	VH11.IdXML					:=	'1';
	VH11.TagXML					:=	4;
	VH11.DEF_On.IdXML			:=	'3';
	VH11.DEF_On.TagXML			:=	2;
	VH11.DEF_Off.IdXML			:=	'3';
	VH11.DEF_Off.TagXML			:=	4;
	VH11.DEF_Sensor.IdXML		:=	'3';
	VH11.DEF_Sensor.TagXML		:=	13;
	VH11.DEF_On_Imposs.IdXML	:=	'3';
	VH11.DEF_On_Imposs.TagXML	:=	6;
	VH11.DEF_Off_Imposs.IdXML	:=	'3';
	VH11.DEF_Off_Imposs.TagXML	:=	9;
	VH11.DEF_Off_auto.IdXML		:=	'3';
	VH11.DEF_Off_auto.TagXML	:=	11;

	VS11.IdXML					:=	'1';
	VS11.TagXML					:=	3;

	VINT.IdXML					:=	'1';
	VINT.TagXML					:=	1;
	VINT.DEF_On.IdXML			:=	'3';
	VINT.DEF_On.TagXML			:=	2;
	VINT.DEF_Off.IdXML			:=	'3';
	VINT.DEF_Off.TagXML			:=	4;
	VINT.DEF_Sensor.IdXML		:=	'3';
	VINT.DEF_Sensor.TagXML		:=	13;
	VINT.DEF_On_Imposs.IdXML	:=	'3';
	VINT.DEF_On_Imposs.TagXML	:=	6;
	VINT.DEF_Off_Imposs.IdXML	:=	'3';
	VINT.DEF_Off_Imposs.TagXML	:=	9;
	VINT.DEF_Off_auto.IdXML		:=	'3';
	VINT.DEF_Off_auto.TagXML	:=	11;


(* Gestion FM et FD régénération*)
FM_REGEN(CLK:=PS11.STATE_Regen);
FD_REGEN(CLK:=PS11.STATE_Regen);
END_ACTION

END_FUNCTION_BLOCK

// ---- POUs/Fonction/FONCTIONS PUISSANCE/BLOCK_CPT_USURE_OLD.TcPOU
FUNCTION_BLOCK BLOCK_CPT_USURE_OLD

VAR_INPUT
	I_Machine_prod:			BOOL;		(*Indicateur de machine en process*)
	I_EVAP_ON:	BOOL;			(*Indicateur d'évaporation en cours*)
END_VAR

VAR
	O_Rapport:					BOOL;		(*demande d'édition du rapport de consommation, c'est l'outil externe qui la fait retomber*)

	FM_Prod:					R_TRIG;		(*Front montant de debut de prod*)
	FM_Layer_Load_Ok:			R_TRIG;		(*Front montant de chargement couche ok*)
	FM_Layer:					R_TRIG;		(*Front montant début évaporation*)
	FD_Prod:					F_TRIG;		(*Front descendant de fin de prod*)

	FD_O_Rapport:				F_TRIG;		(*Front descendant de demande d'édition du rapport*)
	FD_Layer:					F_TRIG;		(*Front descendant de fin de couche*)

	VAR_New_File:				BOOL;		(*Indique si un nouveau fichier doit être créee*)


END_VAR

VAR_OUTPUT
	(*Données du rapport*)
	STATE_User_Login:			STRING[30];	(*Login user ayant lancé la prod*)
	STATE_User_Name:			STRING[30];	(*Nom user ayant lancé la prod*)
	STATE_User_First:			STRING[30];	(*Prénom user ayant lancé la prod*)

	STATE_Process_Name:		STRING;		(*Nom du procédé lancé*)
	STATE_Date_Deb:			DT;			(*Debut du process*)
	STATE_Date_Fin:				DT;			(*Fin du process*)


	STATE_Config:			STRING;		(*Configuration utilisé*)
	STATE_Crucible:			USINT;		(*Numéro du creuset utilisé*)
	STATE_Material:				STRING;		(*Nom du matériau utilisé*)

	STATE_THICK_Consigne:			REAL;	(*Epaisseur saisie par l'utilisateur au début de la recette*)
	STATE_THICK_Obtenue:			REAL;	(*Epaisseur obtenue en fin de couche ou sur arrêt procédé*)

	STATE_Date_Deb_Evap:		DT;		(*Début d'évaporation*)
	STATE_Date_Fin_Evap:		DT;		(*Fin évaporation*)
	STATE_Temps_Depot:			INT;	(*Temps du dépôt*)

END_VAR

(*Gestion des fronts*)
FM_Prod(clk := I_Machine_prod);
FD_Prod(clk := I_Machine_prod);

FM_Layer(clk := I_EVAP_ON );
FD_Layer(clk := I_EVAP_ON);

FD_O_Rapport(clk := O_Rapport);

(*Remise à 0 des valeurs*)
IF FD_O_Rapport.Q THEN
	STATE_Config				:= '';
	STATE_Crucible				:= 0;
	STATE_Material				:= '';
	STATE_THICK_Consigne		:= 0;
	STATE_THICK_Obtenue			:= 0;
END_IF

(*Enregistrement des données en début de process*)
IF FM_Prod.Q THEN
	VAR_New_File					:=	TRUE;
	STATE_User_Login				:=	PRG_USER.ACTU_USER.LOGIN;
	STATE_User_Name				:=	PRG_USER.ACTU_USER.NOM;
	STATE_User_First				:=	PRG_USER.ACTU_USER.PRENOM;

	STATE_Process_Name			:=	EXECPROC.PRM_PROCESS;
	STATE_Date_Deb				:=	PRG_SEC._date;

END_IF


(*Enregistrement des données liées à l'empilement*)
IF FM_Layer_Load_Ok.Q THEN
	STATE_Config				:= PRG_MOUVEMENT_PS.STATE_Dome_Type;
	STATE_Crucible				:= PRG_EVAP.EVAPS1.PRM_NCR;
	STATE_Material				:= PRG_EVAP.CRUCIBLE1.PRM_MAT[STATE_Crucible];
	STATE_THICK_Consigne		:= MAIN.STEP_EMPILEMENT.PRM_EPAISSEUR;
END_IF


(*Enregistrements des données en début de couche*)
IF FM_Layer.Q THEN
	STATE_Date_Deb_Evap				:= PRG_SEC._date;
END_IF


(*Enregistrements des données en fin de couche*)
IF FD_Layer.Q THEN
	STATE_Date_Fin_Evap				:= PRG_SEC._date;
	STATE_THICK_Obtenue			:= MAIN.STEP_EMPILEMENT.STATE_RATE_AGREGATE;

		(*Levée du bit de demande de création d'un nouveau fichier*)
		O_Rapport					:=	TRUE;

END_IF


IF FD_Prod.Q THEN
	STATE_Date_Fin	:= PRG_SEC._date;

		(*Levée du bit de demande de création d'un nouveau fichier*)
		O_Rapport					:=	TRUE;

END_IF

END_FUNCTION_BLOCK

// ---- POUs/Fonction/FONCTIONS SERVITUDES/BLOCK_LIGNE_REF_FLOWTEMP.TcPOU
FUNCTION_BLOCK BLOCK_LIGNE_REF_FLOWTEMP

(* Fonction de gestion d'une ligne d'eau avec débitmètre SV4200 (Vanne avec ou sans débitmètre*)

(****************historique des versions*****************************)
(* Version 1-0 - GV - 07/2023 - VERSION INITIALE - 13905*)
(********************************************************************)

VAR_INPUT
	RESET:					BOOL;
	MANUAL:					BOOL;			(* ~ (OPC : 1 : available for OPC-clients) *)
	DEx:					BLOCK_SV4200;

	CO_On:					BOOL;								(*commande de marche*)
                                                                
	I_Cond_need_Ref:		BOOL;								(*condition qui necessite le refroidissement*)
	I_inhibe_surv_ref:		BOOL;								(*Condition d'inhibition de la surveillance du débit*)
	I_Cond_ref_Ok:			BOOL;								(*Condition de validation du bon refroidissment (Temp, ...) *)
                                                                
	VEx:					BLOCK_ACTUATOR;						(*vanne d'eau simple*)
                                                                
	DEF_Ref:				PRCDEF;								(*défaut de refroidissement*)
	DEF_Dex:				PRCDEF;								(*défaut de fonctionnement du débitmètre*)
	                                                            
	DEF_Low_Flow:			PRCDEF;								(*défaut débit insuffisant*)
	DEF_High_Flow:			PRCDEF;								(*défaut débit trop important*)
	DEF_Low_Temp:			PRCDEF;								(*défaut température trop basse*)
	AL_High_Temp:			PRCDEF;								(*alarme température trop haute*)
	DEF_High_Temp:			PRCDEF;								(*défaut température trop haute*)
END_VAR

VAR_INPUT PERSISTENT
	CONF_NO_DexT:			BOOL;								(*option pas de débitmètre*)
	CONF_TIM_OFF:			TIME;								(* ~ (OPC : 1 : available for OPC-clients) *)		(*temps entre la perte de la condition absolue de refroidissement
																					et la fermeture de la vanne d'eau*)
	CONF_No_Def_Dex:		BOOL;													(*pas de surveillance du défaut de fermeture de la vanne*)

	CONF_Eau_chaude:		BOOL;			(*ligne d'eau raccordée à un circuit eau chaude/froide*)
	
	CONF_Min_Flow:			REAL;			(*débit minimum*)
	CONF_Max_Flow:			REAL;			(*Débit maximum*)
	CONF_Min_Temp:			REAL;			(*Température minimum*)
	CONF_Max_Temp:			REAL;			(*Température maximum pour défaut*)	
	CONF_Max_Temp_AL:		REAL;			(*Température maximum pour alarme*)

	(*Entité*)
	IsAssembly:				BOOL;			(*entité : assemblage*)
	IdXML:					STRING;			(*nom entité : identifiant pour recherche dans dico*)
	TagXML:					UINT;			(*nom entité : identifiant pour recherche dans dico*)
	IdParent:				STRING;			(*MNEMO de l'appelant*)
	MNEMO:					STRING;			(*MNEMO de l'entité*)
	MNEMO_Dex:				STRING;			(*MNEMO du débitmètre*)
END_VAR

VAR_OUTPUT
	STATE_Ok:				BOOL;			(* ~ (OPC : 1 : available for OPC-clients) *)		(*refroidissement ok*)
	STATE_Ar:				BOOL;			(* ~ (OPC : 1 : available for OPC-clients) *)		(*refroidissement à l'arrêt*)
	STATE_NOk:				BOOL;			(* ~ (OPC : 1 : available for OPC-clients) *)		(*refroidissement à l'arrêt*)
	STATE_DexT:				BOOL;			(* ~ (OPC : 1 : available for OPC-clients) *)		(*seuil débitmètre*)
END_VAR

VAR
	TIMER_OFF:					TON;
	VAR_Etape:					USINT;															(*Etape du grafcet de gestion de la servitudes*)
	VAR_DExT:					BOOL;
END_VAR

Def_Ref.IdXML				:=	'8';
Def_Ref.TagXML				:=	1;

DEF_Dex.IdXML				:=	'8';
DEF_Dex.TagXML				:=	2;

DEF_Low_Flow.IdXML			:=	'8';
DEF_Low_Flow.TagXML			:=	15;
DEF_High_Flow.IdXML			:=	'8';
DEF_High_Flow.TagXML		:=	16;
DEF_Low_Temp.IdXML			:=	'8';
DEF_Low_Temp.TagXML			:=	17;
DEF_High_Temp.IdXML			:=	'8';
DEF_High_Temp.TagXML		:=	18;
AL_High_Temp.IdXML			:=	'8';
AL_High_Temp.TagXML			:=	18;
AL_High_Temp.Groupe			:=	1;

VEx.IdParent				:=	MNEMO;
VEx.IdXML					:=	'1';
VEx.TagXML					:=	1;
VEx.DEF_Off_auto.IdXML		:=	'3';
VEx.DEF_Off_auto.TagXML		:=	11;
VEx.DEF_Off_Imposs.IdXML	:=	'3';
VEx.DEF_Off_Imposs.TagXML	:=	9;
VEx.DEF_On_Imposs.IdXML		:=	'3';
VEx.DEF_On_Imposs.TagXML	:=	6;
VEx.DEF_On.IdXML			:=	'3';
VEx.DEF_On.TagXML			:=	2;
VEx.DEF_Off.IdXML			:=	'3';
VEx.DEF_Off.TagXML			:=	4;
VEx.DEF_Sensor.IdXML		:=	'3';
VEx.DEF_Sensor.TagXML		:=	13;
	
(*Débitmètre*)
DEx.RESET		:=	RESET OR CONF_NO_DexT;
DEx();

VAR_DExT := (DEx.STATE_Flow >= CONF_Min_Flow) AND (DEx.STATE_Flow <= CONF_Max_Flow); (*On considère qui il y a du débit si compris entre MIN et MAX*)

(*Défaut débit insufisant*)
DEF_Low_Flow.CONDITION	:=	VEx.OUT_On AND DEx.STATE_OK AND NOT CONF_NO_DexT AND (DEx.STATE_Flow < CONF_Min_Flow) AND (CONF_Min_Flow <> 0) AND NOT RESET;
DEF_Low_Flow.VAL1		:=	CONCAT(REAL_TO_STRING(CONF_Min_Flow),'L/min /');
DEF_Low_Flow.VAL1		:=	CONCAT(DEF_Low_Flow.VAL1,TIME_TO_STRING(DEF_Low_Flow.DELAY));
DEF_Low_Flow();
(*Défaut débit trop important*)
DEF_High_Flow.CONDITION	:=	VEx.OUT_On AND DEx.STATE_OK AND NOT CONF_NO_DexT AND (DEx.STATE_Flow > CONF_Max_Flow) AND (CONF_Max_Flow <> 0) AND NOT RESET;
DEF_High_Flow.VAL1		:=	CONCAT(REAL_TO_STRING(CONF_Max_Flow),'L/min /');
DEF_High_Flow.VAL1		:=	CONCAT(DEF_High_Flow.VAL1,TIME_TO_STRING(DEF_High_Flow.DELAY));
DEF_High_Flow();
(*Défaut température trop basse*)
DEF_Low_Temp.CONDITION	:=	VEx.OUT_On AND DEx.STATE_OK AND NOT CONF_NO_DexT AND (DEx.STATE_Temp < CONF_Min_Temp) AND NOT RESET;
DEF_Low_Temp.VAL1		:=	CONCAT(REAL_TO_STRING(CONF_Min_Temp),'°C/');
DEF_Low_Temp.VAL1		:=	CONCAT(DEF_Low_Temp.VAL1,TIME_TO_STRING(DEF_Low_Temp.DELAY));
DEF_Low_Temp();
(*Défaut température trop haute*)
DEF_High_Temp.CONDITION	:=	VEx.OUT_On AND DEx.STATE_OK AND NOT CONF_NO_DexT AND (DEx.STATE_Temp > CONF_Max_Temp) AND NOT RESET;
DEF_High_Temp.VAL1		:=	CONCAT(REAL_TO_STRING(CONF_Max_Temp),'°C/');
DEF_High_Temp.VAL1		:=	CONCAT(DEF_High_Temp.VAL1,TIME_TO_STRING(DEF_High_Temp.DELAY));
DEF_High_Temp();
(*Alarme température trop importante*)
AL_High_Temp.CONDITION	:=	VEx.OUT_On AND DEx.STATE_OK AND NOT CONF_NO_DexT AND (DEx.STATE_Temp > CONF_Max_Temp_AL) AND NOT RESET;
AL_High_Temp.VAL1		:=	CONCAT(REAL_TO_STRING(CONF_Max_Temp_AL),'°C/');
AL_High_Temp.VAL1		:=	CONCAT(AL_High_Temp.VAL1,TIME_TO_STRING(AL_High_Temp.DELAY));
AL_High_Temp();

(* initialisation du grafcet*)
IF 		VAR_etape = 0
		THEN
				VAR_etape.0 := TRUE;
(*repositionnement sur étape 0*)
ELSIF	MANUAL OR RESET
		THEN
				VAR_etape := 0;				(*RAZ grafcet*)
				VAR_etape.0:= TRUE;
(*étape 0-1*)
ELSIF 	VAR_etape.0
		AND CO_On
		THEN
				VAR_etape.1:= TRUE;
				VAR_etape.0:= FALSE;
(*étape 1-0*)
ELSIF 	VAR_etape.1
		AND NOT CO_on AND TIMER_OFF.Q
		THEN
				VAR_etape.0:= TRUE;
				VAR_etape.1:= FALSE;
END_IF;

(*Traitement en sortie*)
TIMER_OFF.PT	:=	CONF_TIM_OFF;
TIMER_OFF.IN	:=	VAR_Etape.1 AND NOT CO_On;
TIMER_OFF();

(*bit d'état*)
IF		((VAR_Etape.1 AND ((VAR_DExT AND DEx.STATE_OK) OR CONF_NO_DExT) AND NOT MANUAL AND VEx.OUT_On)
		OR (MANUAL AND ((VAR_DExT AND DEx.STATE_OK) OR CONF_NO_DExT)  AND VEx.OUT_On)) 
			AND I_Cond_ref_Ok AND NOT DEF_Low_Temp.DEF AND NOT DEF_High_Temp.DEF THEN
	STATE_Ok	:=	TRUE;
ELSIF	(NOT VAR_Etape.1 AND NOT MANUAL)
		OR DEF_Ref.DEF OR DEF_Low_Temp.DEF OR DEF_High_Temp.DEF
		OR (MANUAL AND NOT (VAR_DExT AND DEx.STATE_OK) AND NOT CONF_NO_DExT AND VEx.OUT_On)
		OR NOT VEx.OUT_On
		OR NOT I_Cond_ref_Ok THEN
	STATE_Ok	:=	FALSE;
END_IF
STATE_Ar		:=	(VAR_Etape.0 AND NOT MANUAL) OR (MANUAL AND NOT VEx.OUT_ON) OR RESET;
STATE_NOk		:=	DEF_Dex.DEF OR DEF_Ref.DEF OR DEF_High_Flow.DEF OR DEF_High_Temp.DEF OR DEF_Low_Flow.DEF OR DEF_Low_Temp.DEF OR (DEx.STATE_NOK AND NOT CONF_NO_DexT);
STATE_DexT		:=  (VAR_DExT OR CONF_NO_DexT);


(*Pilotage de la vanne*)
VEx(
	RESET:=					RESET ,
	MANUAL:=				MANUAL ,
	CO_On:=					VAR_Etape.1,
	CONF_EN_On:= 			1,
	CONF_No_Safety_Auto:=	0,
	CONF_Tim_Valid_On:=		T#200ms,
	CONF_Tim_Valid_Off:= 	T#200ms);


(*Défaut de refroidissement*)
DEF_Ref.CONDITION		:=	VEx.OUT_On AND NOT VAR_DExT AND NOT CONF_NO_DexT AND NOT RESET
							AND NOT I_Inhibe_Surv_Ref;
DEF_Ref();

(*Défaut débitmètre ou fermeture vanne*)
DEF_DEx.CONDITION		:=	NOT VEx.OUT_On AND VAR_DExT AND NOT CONF_No_Def_Dex AND NOT RESET AND NOT CONF_NO_DexT;
DEF_DEx.DELAY			:= 	T#60s;
DEF_DEx();

END_FUNCTION_BLOCK

// ---- TextLists/GlobalTextList.TcGTLO
TEXTLIST GlobalTextList
  502 = ' '
  2160 = '                                                                                                                                                                                                                                                                                                                                                                                                                                                   '
  950 = '  SOURCE 1'
  404 = ' %.1f %%'
  75 = ' %1.0'
  76 = ' %1.0f'
  74 = ' %1.0f %%'
  78 = ' %1.0f Hz'
  73 = ' %1.0f V'
  77 = ' %1.0fHz'
  71 = ' %1.1f %%'
  2347 = ' %1.1f A'
  140 = ' %1.1f mA '
  175 = ' %1.1f rpm'
  615 = ' %1.1f tr/min'
  2064 = ' %1.1f V'
  1485 = ' %1.2f'
  144 = ' %1.2f A'
  80 = ' %1.2f A°/s'
  1182 = ' %1.2f KV'
  79 = ' %1.2fA°/s'
  143 = ' %1.3f kA°'
  919 = ' %1.3f MHz'
  831 = ' %2.0f °/s2'
  172 = ' %2.2f mmps'
  822 = ' %2.2f rpm'
  171 = ' %3.1f mm'
  826 = ' %3.1f °'
  2275 = ' %i s'
  103 = ' %s'
  1278 = ' / '
  857 = ' CONF_MAX_TORQUE'
  2574 = ' CONF_PMax'
  1444 = ' Creuset'
  93 = ' DEF_PPrim.DELAY'
  88 = ' DEF_TGF.DELAY'
  94 = ' DEF_Vent.DELAY'
  2073 = ' In: %1.2f A'
  1450 = ' Matériau'
  33 = ' mbar' | FR: 'mbar' | EN: 'mbar'
  2030 = ' ON'
  735 = ' P'
  34 = ' Pa' | FR: 'Pa' | EN: 'Pa'
  1083 = ' PRM_Adresse_IP_XTC'
  837 = ' PRM_DEC'
  2565 = ' PRM_Max_Temp'
  89 = ' PRM_Pr_Atm'
  91 = ' PRM_Pr_PPrim'
  92 = ' PRM_Pr_RP_PPrim'
  87 = ' PRM_Pr_TGF'
  130 = ' PRM_Pr_Trf_CH'
  131 = ' PRM_Pr_Trf_LL'
  846 = ' PRM_SURV_VROT'
  97 = ' PRM_Th_Life'
  1104 = ' PRM_Tim_Ala_Pr'
  572 = ' PRM_Tim_Def_Pr'
  90 = ' PRM_Tim_SurVentil_E'
  849 = ' PRM_TIM_SURV_VROT'
  443 = ' PRM_tps_att_chaud'
  680 = ' PRM_Tp_Vent'
  536 = ' Ta'
  1100 = ' Ta (s)'
  2170 = ' Td'
  1097 = ' Td (s)'
  662 = ' Ti'
  1093 = ' Ti (s)'
  32 = ' Torr' | FR: 'Torr' | EN: 'Torr'
  174 = ' Vitesse:'
  343 = '"%t[HH:mm:ss]"'
  1339 = '%.1f A'
  3230 = '%.1f l/s'
  853 = '%.1f N'
  1040 = '%.1f sccm'
  1333 = '%.1f V'
  393 = '%.1f °C'
  2195 = '%.2f A'
  58 = '%.2f kV'
  59 = '%.3f %%'
  169 = '%1.0f'
  1567 = '%1.0f %'
  99 = '%1.0f %%'
  535 = '%1.0f K'
  2414 = '%1.0f mA'
  72 = '%1.0f mA '
  811 = '%1.0f rpm'
  1499 = '%1.0f V'
  903 = '%1.0f °C'
  31 = '%1.1e'
  112 = '%1.1e mbar'
  114 = '%1.1e mbar.L/s'
  113 = '%1.1f'
  189 = '%1.1f '
  142 = '%1.1f %%'
  86 = '%1.1f L'
  931 = '%1.1f l/s'
  70 = '%1.1f mA'
  125 = '%1.1f mm'
  126 = '%1.1f mm/s'
  1644 = '%1.1f mmps'
  1657 = '%1.1f rpm'
  618 = '%1.1f tr/min'
  537 = '%1.1f V'
  968 = '%1.1f °'
  138 = '%1.1f °C'
  3068 = '%1.1f%'
  653 = '%1.1f%%'
  65 = '%1.2e mbar'
  134 = '%1.2f'
  55 = '%1.2f %%'
  845 = '%1.2f KV '
  935 = '%1.2f rpm'
  940 = '%1.2f °'
  68 = '%1.2f Å/s'
  135 = '%1.3f'
  67 = '%1.3f kÅ'
  841 = '%2.2f rpm'
  3428 = '%3.0f'
  726 = '%3.1f'
  833 = '%3.2f °'
  782 = '%4.0f'
  664 = '%4.1f'
  665 = '%4.1f '
  870 = '%4.2f'
  1889 = '%c'
  342 = '%d'
  45 = '%i'
  136 = '%i '
  137 = '%i     '
  160 = '%i %'
  161 = '%i %%'
  133 = '%i mm'
  148 = '%i s'
  1621 = '%m'
  1 = '%s' | FR: '%s' | EN: '%s'
  1443 = '%S'
  699 = '%s '
  1296 = '%s  '
  2128 = '%s (%)'
  2287 = '%s (Hz)'
  2041 = '%s (MHz)'
  438 = '%s :'
  101 = '%s s'
  3884 = '%s sec'
  527 = '%t'
  638 = '%t%H%M%S'
  1107 = '%t%x'
  2402 = '%t(%H%M%S)'
  1769 = '%t[%H%M%S]'
  1423 = '%t[%H:%M:%S]'
  1134 = "%t[h'h''m'm's's'ms'ms']"
  224 = "%t[h'h'm'm's's'ms'ms']"
  2932 = '%t[HH:MM:MS]'
  813 = '%t[HH:mm:ss:ms]'
  1128 = '%t[HH:mm:ss]'
  2695 = '%t[HH:MM:SS]'
  1686 = "%t[m'm's's']"
  2850 = '%t[s]'
  1459 = '%x'
  247 = '+'
  154 = '+0.1%'
  158 = '+0.1%%'
  155 = '+1%'
  159 = '+1%%'
  637 = '-'
  153 = '-0.1%'
  157 = '-0.1%%'
  152 = '-1%'
  156 = '-1%%'
  180 = '.1'
  181 = '.2'
  121 = '/'
  104 = '1'
  105 = '2'
  3 = '22222'
  106 = '3'
  107 = '4'
  108 = '5'
  109 = '6'
  110 = '7'
  111 = '8'
  42 = '?' | FR: '?' | EN: '?'
  29 = '??????' | FR: '??????' | EN: '??????'
  2017 = 'Ack'
  168 = 'Activity'
  0 = 'Adresse Alliance ' | FR: '4 Avenue du Pont de Tasset - 74960 CRAN GEVRIER - FRANCE\ntel: +33 (0)4 50 57 93 85 - fax: +33 (0)4 50 57 96 74\nurl: http://www.alliance-concept.com - mail: contact@alliance-concept.com' | EN: '4 Avenue du Pont de Tasset - 74960 CRAN GEVRIER - FRANCE\ntel: +33 (0)4 50 57 93 85 - fax: +33 (0)4 50 57 96 74\nurl: http://www.alliance-concept.com - mail: contact@alliance-concept.com'
  673 = 'ALM_SURV.DELAY'
  2747 = 'ALM_SURV.OFFSET'
  3220 = 'ALM_SURV_CURRENT.DELAY'
  887 = 'ALM_SURV_CURRENT.OFFSET'
  3226 = 'ALM_SURV_VOLTAGE.DELAY'
  2512 = 'ALM_SURV_VOLTAGE.OFFSET'
  5 = 'Annuler' | FR: 'Annuler' | EN: 'Cancel'
  2056 = 'Anode : %1.1f A '
  40 = 'AUTO'
  27 = 'BALAYAG' | FR: 'BALAYAGE' | EN: 'SWEEPING'
  173 = 'Balayage'
  3154 = 'BALAYAGE'
  2068 = 'Balayage :'
  2039 = 'BEAM'
  66 = 'Bouton_navig'
  116 = 'Cache' | FR: 'Cache :' | EN: 'Shutter:'
  117 = 'Cache %s' | FR: 'Cache : %s' | EN: 'Shutter: %s'
  2403 = 'Cancel'
  56 = 'CANON'
  383 = 'CANON e-'
  1327 = 'CANON_ION'
  82 = 'chambre Ouvert' | FR: 'Chambre ouverte' | EN: 'Open chamber'
  1187 = 'Chambre Ouverte'
  1033 = 'CHRONO'
  28 = 'CLAPET_MANU'
  22 = 'Conf.' | FR: 'Config.' | EN: 'Sett.'
  3155 = 'CONFIG_CHAUFFAGE_PARAM'
  445 = 'CONFIG_ETUVAGE_PARAM'
  1088 = 'CONFIG_EVAP_PARAM'
  178 = 'CONFIG_IAD_INFOS'
  829 = 'CONFIG_PS_PARAM'
  1159 = 'CONFIG_TITRE_PS'
  84 = 'CONFIG_TPS_INFOS' | FR: 'Format temps : T#0h0m0s0ms' | EN: 'Time format: T#0h0m0s0ms'
  333 = 'CONF_Courant_Plasma'
  146 = 'CONF_Evap_Cont'
  150 = 'CONF_Maximum_Time'
  162 = 'CONF_Maximum_Time_S1'
  163 = 'CONF_Maximum_Time_S2'
  1710 = 'CONF_Max_Flow'
  1750 = 'CONF_Max_Temp'
  1965 = 'CONF_Max_Temp_Al'
  825 = 'CONF_Max_Temp_IN'
  2305 = 'CONF_Max_Temp_OUT'
  1136 = 'CONF_Min_Flow'
  1465 = 'CONF_Min_Temp'
  179 = 'CONF_Min_Temp_IN'
  2551 = 'CONF_Min_Temp_OUT'
  139 = 'CONF_No_Mvts_In_Process'
  149 = 'CONF_RateWatcher_Acc'
  147 = 'CONF_RateWatcher_Time'
  1074 = 'CONF_Temp_Max'
  1283 = 'CONF_Temp_Min'
  1525 = 'CONF_Tension_Plasma'
  2251 = 'CONF_Tps_Pompage_Theorique'
  431 = 'Consigne'
  1627 = 'Courant'
  1032 = 'Creuset'
  3009 = 'CREUSET'
  3019 = 'CREUSET_STATE'
  164 = 'Crsytal'
  2443 = 'CRUCIBLE : %s'
  830 = 'Cryo'
  165 = 'Crystal'
  24 = 'Créer' | FR: 'Créer' | EN: 'Create'
  13 = 'Créer...' | FR: 'Créer...' | EN: 'Create...'
  62 = 'Current' | FR: 'Courant' | EN: 'Current'
  145 = 'D'
  2782 = 'DEF_SURV.DELAY'
  463 = 'DEF_SURV.OFFSET'
  1378 = 'DEF_SURV_CURRENT.DELAY'
  1544 = 'DEF_SURV_CURRENT.OFFSET'
  2659 = 'DEF_SURV_VOLTAGE.DELAY'
  672 = 'DEF_SURV_VOLTAGE.OFFSET'
  30 = 'Degas' | FR: 'Degaz' | EN: 'Degas'
  406 = 'delay'
  47 = 'ENGLISH' | FR: 'ENGLISH' | EN: 'ENGLISH'
  141 = 'EXIT' | FR: 'Quitter' | EN: 'EXIT'
  177 = 'FAIL'
  16 = 'Fermer' | FR: 'Fermer' | EN: 'Close'
  23 = 'FoncSA.' | FR: 'Fonc. Av.' | EN: 'Adv. func.'
  46 = 'FRANCAIS' | FR: 'FRANCAIS' | EN: 'FRANCAIS'
  167 = 'Freq. (Hz)'
  2481 = 'Gaz'
  2509 = 'Gaz 1'
  1501 = 'Gaz 2'
  772 = 'GO'
  12 = 'Groupe' | FR: 'Groupe' | EN: 'Group'
  806 = 'Haute Tension'
  60 = 'HighVolt' | FR: 'Haute tension' | EN: 'High voltage'
  124 = 'Homed' | FR: 'Homed' | EN: 'Homed'
  1036 = 'IAD_SA'
  176 = 'IC6'
  676 = 'IC6_SA'
  2 = 'IDClient:%s' | FR: 'Client : %s' | EN: 'Customer: %s'
  9 = 'Identifiant' | FR: 'Identifiant' | EN: 'Login'
  2047 = 'Ie: %1.1f A'
  1990 = 'Info'
  120 = 'INFO_PROCESS_BOUTON'
  119 = 'INFO_PROCESS_VISU'
  1163 = 'load'
  53 = 'LOCAL' | FR: 'LOCAL' | EN: 'LOCAL'
  613 = 'M'
  64 = 'M11 :'
  69 = 'M12 :'
  128 = 'M21 :'
  129 = 'M21:'
  19 = 'Maint.' | FR: 'Maint.' | EN: 'Maint.'
  1585 = 'maintenance cryo'
  41 = 'MANUEL'
  1901 = 'Matériau source 2'
  1907 = 'Matériau source 3'
  83 = 'MENU_CONFIG_FONC'
  183 = 'mode'
  44 = 'MODE_AUTO' | FR: 'Automatique' | EN: 'Automatic'
  43 = 'MODE_MANUEL' | FR: 'Manuel' | EN: 'Manual'
  7 = 'Modifier' | FR: 'Modifier' | EN: 'Modify'
  14 = 'Modifier...' | FR: 'Modifier...' | EN: 'Modify...'
  115 = 'Motif' | FR: 'Motif :' | EN: 'Pattern:'
  1212 = 'm_input_IAD.'
  57 = 'NOK'
  10 = 'Nom' | FR: 'Nom' | EN: 'Last name'
  17 = 'Nom du groupe' | FR: 'Nom du groupe' | EN: 'Group Name'
  1947 = 'NOM_VERIN'
  8 = 'Non' | FR: 'Non' | EN: 'No'
  2268 = 'N°'
  49 = 'OFF' | FR: 'OFF' | EN: 'OFF'
  557 = 'Off'
  4 = 'OK' | FR: 'OK' | EN: 'OK'
  122 = 'OK!'
  48 = 'ON' | FR: 'ON' | EN: 'ON'
  2657 = 'On'
  25 = 'OPTIONS' | FR: 'OPTIONS' | EN: 'OPTIONS'
  6 = 'Oui' | FR: 'Oui' | EN: 'Yes'
  81 = 'Ouvert'
  341 = 'Pompage'
  170 = 'POMPAGE'
  63 = 'Power' | FR: 'Puissance' | EN: 'Power'
  11 = 'Prenom' | FR: 'Prénom' | EN: 'First name'
  1458 = 'PRG_DEF_MANAGEMENT.EVENT_LIST[INDEX].STATE_dt'
  429 = 'PRM_Border_Ratio'
  102 = 'PRM_Fact_Surv_Dep'
  368 = 'PRM_Max_Tim_W'
  311 = 'PRM_Pr_Canon_ion_Ok'
  132 = 'PRM_Pr_Canon_Ok'
  98 = 'PRM_Th_Life'
  346 = 'PRM_Tim_Ala_Pr'
  629 = 'PRM_Tim_Bal_BalInt'
  1020 = 'PRM_Tim_Def_Pr'
  2971 = 'PRM_Tim_FinBal'
  932 = 'PRM_Tim_Int_BalInt'
  100 = 'PRM_Tim_Surv_Dep'
  51 = 'Pro\nfUNC' | FR: 'Fonctions\nProcess' | EN: 'Process\nFuctions'
  18 = 'Pro. Ed' | FR: 'Ed. proc.' | EN: 'Proc. ed.'
  21 = 'Prod.' | FR: 'Prod.' | EN: 'Prod.'
  118 = 'PRODUCTION' | FR: 'PRODUCTION' | EN: 'PRODUCTION'
  755 = 'PS'
  52 = 'pUMP\nFUNC' | FR: 'Fonctions\nPompage' | EN: 'Pumping\nFunctions'
  1589 = 'Pump TC'
  26 = 'Quitter' | FR: 'Quitter' | EN: 'Exit'
  166 = 'Rate (A/s)'
  54 = 'RDY' | FR: 'RDY' | EN: 'RDY'
  1176 = 'Regen'
  50 = 'REMOTE' | FR: 'REMOTE' | EN: 'REMOTE'
  1090 = 'Remote'
  3704 = 'Retour'
  3029 = 'Rotation'
  123 = 'sas Ouvert' | FR: 'Sas ouvert' | EN: 'Open loadlock'
  666 = 'sccm'
  679 = 'SD11'
  151 = 'Ss'
  977 = 'Start'
  1472 = 'Start / Stop'
  2044 = 'Start/Stop'
  1279 = 'STOP'
  1626 = 'Stop'
  2215 = 'STOP PROCESS'
  61 = 'Stp' | FR: 'Consigne' | EN: 'Setpoint'
  20 = 'Superv.' | FR: 'Admin.' | EN: 'Admin.'
  15 = 'Supprimer' | FR: 'Supprimer' | EN: 'Delete'
  1291 = 'TRAC Record'
  1937 = 'VANNE_CONF'
  1931 = 'VANNE_MODE'
  1956 = 'VERIN_MANU'
  37 = 'Vers Visu manu'
  38 = 'Vers Visu manu\navec placeholder'
  39 = 'Vers Visu standard'
  36 = 'Vesr Visu manu'
  85 = 'Volume' | FR: 'Volume' | EN: 'Volume'
  95 = 'Volume chambre' | FR: 'Volume chambre' | EN: 'Chamber volume'
  96 = 'Volume sas' | FR: 'Volume sas' | EN: 'Loadlock volume'
  127 = 'WithHome' | FR: 'Avec PO' | EN: 'With Homing'
  35 = 'X'
  2302 = 'XTAL6'
  1500 = 'ùs'
END_TEXTLIST

// ---- TextLists/TextList_1Run_1Quartz.TcTLO
TEXTLIST TextList_1Run_1Quartz
  0 = '1 Run = 1 Quartz' | FR: '1 Run = 1 Quartz' | EN: '1 Run = 1 Quartz'
  1 = 'yes' | FR: 'Activé' | EN: 'Activated'
  2 = 'no' | FR: 'Désactivé' | EN: 'Disabled'
  3 = 'raz' | FR: 'Forcage changement quartz' | EN: 'Quartz change forcing'
  4 = 'next' | FR: 'Quartz prévu pour le prochain run' | EN: 'Scheduled quartz for next run'
  5 = 'change' | FR: 'Changement de tous les quartz\n\nnécessaire pour le prochain run' | EN: 'Change all quartz is needed\n\nfor next run'
   = ''
END_TEXTLIST

// ---- TextLists/TextList_Actuator_Type.TcTLO
TEXTLIST TextList_Actuator_Type
  0 = '' | FR: 'Vérin de clampage' | EN: 'Clamping jack'
   = ''
END_TEXTLIST

// ---- TextLists/TextList_Basiques.TcTLO
TEXTLIST TextList_Basiques
  0 = 'OK' | FR: 'OK' | EN: 'OK'
  1 = 'Annul' | FR: 'Annuler' | EN: 'Cancel'
  2 = 'Modifier' | FR: 'Modifier' | EN: 'Modify'
  3 = 'Oui' | FR: 'Oui' | EN: 'Yes'
  4 = 'Non' | FR: 'Non' | EN: 'No'
  5 = 'Créer...' | FR: 'Créer...' | EN: 'Create...'
  6 = 'Modifier...' | FR: 'Modifier...' | EN: 'Modify...'
  7 = 'Supprimer' | FR: 'Supprimer' | EN: 'Delete'
  8 = 'Fermer' | FR: 'Fermer' | EN: 'Close'
  9 = 'Nom' | FR: 'Nom' | EN: 'Name'
  10 = 'Prénom' | FR: 'Prénom' | EN: 'First name'
  11 = 'Créer' | FR: 'Créer' | EN: 'Create'
  12 = 'OPTIONS' | FR: 'OPTIONS' | EN: 'OPTIONS'
  13 = 'Mode_Manuel' | FR: 'Manuel' | EN: 'Manual'
  14 = 'Mode_Auto' | FR: 'Automatique' | EN: 'Automatic'
  15 = 'res' | FR: 'RESET' | EN: 'RESET'
  16 = 'Transfert' | FR: 'Transfert' | EN: 'Transfer'
  17 = 'ch ouvert' | FR: 'Chambre ouverte' | EN: 'Chamber open'
  18 = 'sas ouvert' | FR: 'Sas ouvert' | EN: 'Loadlock open'
  19 = 'modif en ligne' | FR: 'Modification\nen ligne' | EN: 'Online\nmodification'
  22 = 'durée rampe' | FR: 'Durée rampe :' | EN: 'Ramp duration:'
  20 = 'Trac absent' | FR: "ATTENTION : Le logiciel de traçabilité n'est pas lancé! Lancez TrAC" | EN: 'WARNING: Traceability software is not started! Start TrAC'
  21 = 'ACSoft absent' | FR: "ATTENTION : Le logiciel de gestion des évènements n'est pas lancé! Lancez ACSoftware" | EN: 'WARNING: Event logger software is not started! Start ACSoftware'
   = ''
END_TEXTLIST

// ---- TextLists/TextList_Canne_Transfert.TcTLO
TEXTLIST TextList_Canne_Transfert
  0 = 'Canne\t' | FR: 'Canne de transfert' | EN: 'Transfer arm'
  1 = 'Position' | FR: 'Position' | EN: 'Position'
  2 = 'Speed' | FR: 'Vitesse' | EN: 'Speed'
  3 = 'Poste' | FR: 'Position correspondante' | EN: 'Corresponding position'
  4 = 'Poste choisi' | FR: 'Position sélectionnée' | EN: 'Selected position'
  5 = 'Distance' | FR: 'Distance' | EN: 'Distance'
  6 = 'vitesse' | FR: 'Vitesse' | EN: 'Speed'
  7 = 'controle' | FR: 'Opération' | EN: 'Operation'
  8 = 'Durée' | FR: 'Durée : ' | EN: 'Duration:'
  9 = 'ecoulée' | FR: 'Durée écoulée :' | EN: 'Elapsed time:'
   = ''
END_TEXTLIST

// ---- TextLists/TextList_Chauffage.TcTLO
TEXTLIST TextList_Chauffage
  0 = 'chauffage' | FR: 'CHAUFFAGE' | EN: 'HEATING'
  1 = 'puissance' | FR: 'Puissance' | EN: 'Power'
  2 = 'temp' | FR: 'Température' | EN: 'Temperature'
  3 = 'cons temp' | FR: 'Consigne\ntempérature' | EN: 'Temperature\nsetpoint'
  4 = 'cons puiss' | FR: 'Consigne\npuissance' | EN: 'Power\nsetpoint'
  5 = 'cons temp' | FR: 'Consigne temp.' | EN: 'Temp. setpoint'
  6 = 'maintien' | FR: 'Durée de maintien' | EN: 'Hold time'
  7 = 'delta' | FR: 'Variation de temp.' | EN: 'Temp. variation'
  8 = 'max stab' | FR: 'Durée max. de stabilisation' | EN: 'Max. stabilization time'
  9 = 'cons temp' | FR: 'Consigne température' | EN: 'Temperature setpoint'
  10 = 'delta' | FR: 'Variation de température' | EN: 'Temperature variation'
  11 = 'puissance bords' | FR: 'Puissance bords' | EN: 'Borders power'
  12 = 'Tc Ctrl' | FR: 'Thermocouples de régulation' | EN: 'Regulation thermocouples'
  13 = 'Tc Disp' | FR: 'Thermocouples de sécurité' | EN: 'Security thermocouples'
   = ''
END_TEXTLIST

// ---- TextLists/TextList_Config_Chauffage.TcTLO
TEXTLIST TextList_Config_Chauffage
  0 = 'chauffage' | FR: 'CHAUFFAGE' | EN: 'HEATING'
  1 = 'PRM_Tp_Vent' | FR: 'Température max. pour ventilation enceinte' | EN: 'Max. temperature for chamber venting'
  2 = 'PRM_Max_Temp' | FR: 'Consigne température max.' | EN: 'Max. temperature setpoint'
  3 = 'CONF_Pmax' | FR: 'Puissance de chauffage max.' | EN: 'Max. heating setpoint'
  4 = 'P' | FR: 'Gain' | EN: 'Amplification factor'
  5 = 'Ti' | FR: "Temps d'action intégrale" | EN: 'Integral action time'
  6 = 'Td' | FR: "Temps d'action dérivée" | EN: 'Derivative action time'
  7 = 'Ta' | FR: "Temps d'amortissement" | EN: 'Damping time'
  8 = 'PRM_Border_Ratio' | FR: 'Coefficient de pondération chauffage bords' | EN: 'Border heating ratio'
  9 = 'Disable SD11' | FR: 'Désactivation thermocouple SD11' | EN: 'Disable SD11 thermocouple '
  10 = 'Disable SD12' | FR: 'Désactivation thermocouple SD12' | EN: 'Disable SD12 thermocouple '
  11 = 'Disable SD13' | FR: 'Désactivation thermocouple SD13' | EN: 'Disable SD13 thermocouple '
  12 = 'Disable SD14' | FR: 'Désactivation thermocouple SD14' | EN: 'Disable SD14 thermocouple '
  13 = 'Tc Ctrl' | FR: 'Thermocouples de régulation' | EN: 'Regulation thermocouples'
  14 = 'Tc Disp' | FR: 'Thermocouples de sécurité' | EN: 'Security thermocouples'
  15 = 'Tc conf' | FR: 'Configuration thermocouples' | EN: 'Thermocouples settings'
  16 = 'Temp min' | FR: 'Température min. avand défaut' | EN: 'Min. temperature before fault'
  17 = 'Temp max' | FR: 'Température max. avant défaut' | EN: 'Max temperature before fault'
  18 = 'Rechauf' | FR: 'Thermaliseur' | EN: 'Chiller'
   = ''
END_TEXTLIST

// ---- TextLists/TextList_Config_EFFLUVAGE.TcTLO
TEXTLIST TextList_Config_EFFLUVAGE
  0 = 'Effluvage' | FR: 'EFFLUVAGE' | EN: 'GLOW DISCHARGE'
  1 = 'PRM_Tp_Vent' | FR: 'Température max. pour ventilation enceinte' | EN: 'Max. temperature for chamber venting'
  2 = 'PRM_Max_Temp' | FR: 'Consigne température max.' | EN: 'Max. temperature setpoint'
  3 = 'CONF_Pmax' | FR: 'Puissance max.' | EN: 'Max. setpoint'
  4 = 'P' | FR: 'Gain' | EN: 'Amplification factor'
  5 = 'Ti' | FR: "Temps d'action intégrale" | EN: 'Integral action time'
  6 = 'Td' | FR: "Temps d'action dérivée" | EN: 'Derivative action time'
  7 = 'Ta' | FR: "Temps d'amortissement" | EN: 'Damping time'
  8 = 'Tc Ctrl' | FR: 'Seuil de courant de détéction du plasma' | EN: 'Plasma current detection threshold'
  9 = 'Tc Disp' | FR: 'Seuil de tension de détéction du plasma' | EN: 'Plasma voltage detection threshold'
  10 = 'Alimentation' | FR: 'ALIMENTATION' | EN: 'POWER SUPPLY'
  11 = 'alm surv delay' | FR: 'Temps de surveillance avant alarme' | EN: 'Delay before alarm'
  12 = 'alm surv offset' | FR: 'Offset de surveillance avant alarme' | EN: 'Offset before alarm'
  13 = 'dft surv delay' | FR: 'Temps de surveillance avant défaut' | EN: 'Delay before fault'
  14 = 'dft surv offset' | FR: 'Offset de surveillance avant défaut' | EN: 'Offset before fault'
   = ''
END_TEXTLIST

// ---- TextLists/TextList_Config_Evap.TcTLO
TEXTLIST TextList_Config_Evap
  0 = 'reg quartz' | FR: 'Réglage quartz' | EN: 'Crystal setting'
  1 = 'life seuil' | FR: "Seuil d'alarme vie des quartz" | EN: 'Crystal life alarm threshold'
  2 = 'evap settings' | FR: 'Réglages surveillance temps maximum de dépôt' | EN: 'Maximum evaporation time monitoring settings'
  3 = 'prm_tim_surv_dep_min' | FR: 'Temps maximum définissant un dépôt court\nTemps ajouté au temps théorique pour les dépôts courts' | EN: 'Maximum time to determinate a short deposit\nTheorical additional time for short deposit'
  4 = 'PRM_Fact_Surv_Dep' | FR: 'Pourcentage temps supplémentaire ajouté pour les dépôts longs' | EN: 'Additional time porcentage for long deposit'
  5 = 'reg source 1' | FR: 'Réglages source 1' | EN: 'Source 1 settings'
  6 = 'reg source 2' | FR: 'Réglages source 2' | EN: 'Source 2 settings'
  7 = 'matériau' | FR: 'Matériau' | EN: 'Material'
  8 = 'Nom balayage' | FR: 'Nom du balayage' | EN: 'Sweeping name'
  9 = 'no mvts in proc' | FR: 'Inhibition des mouvements canne en process' | EN: 'No transfer arm movements in process'
  10 = 'reglages mvts' | FR: 'Réglages mouvements' | EN: 'Movement settings'
  11 = 'evap continue' | FR: 'Mode évaporation continue' | EN: 'Continuous evaporation mode'
  12 = 'mode actif' | FR: 'Mode évaporation continue actif (si non, mode couche classique)' | EN: 'Continuous evaporation mode active (if not, classical layer mode)'
  13 = 'rate watcher time' | FR: "Interval de temps entre les périodes d'échantillonage" | EN: 'Time interval between sample periods'
  14 = 'rate watcher accuracy' | FR: "Tolérance de la fenêtre de validation de la vitesse d'évaporation" | EN: 'Acceptance window for evaporation rate'
  15 = 'maximum time' | FR: "Temps maximum d'évaporation continue avant arrêt automatique" | EN: 'Maximum time for continuous evaporation before automatic stop'
  16 = 'confirm refill' | FR: 'Cliquez ici pour confirmer que les creusets ont été chargés' | EN: 'Click here to confirm crucible refilling'
  17 = 'maximum time s1' | FR: "Temps maximum d'évaporation continue avant arrêt automatique (Canon 1)" | EN: 'Maximum time for continuous evaporation before automatic stop (E-Gun 1)'
  18 = 'maximum time s2' | FR: "Temps maximum d'évaporation continue avant arrêt automatique (Source Joule)" | EN: 'Maximum time for continuous evaporation before automatic stop (Thermal source)'
  19 = 'maximum time s3' | FR: "Temps maximum d'évaporation continue avant arrêt automatique (Canon 2)" | EN: 'Maximum time for continuous evaporation before automatic stop (E-Gun 2)'
  20 = 'Reg XTC' | FR: 'Réglage XTC' | EN: 'XTC Setting'
  21 = 'IP' | FR: "Adresse IP de l'XTC" | EN: 'Ip Adress of XTC'
  22 = 'Cr' | FR: 'Creuset' | EN: 'Crucible'
  23 = 'CONF_Min_Temp_IN' | FR: 'Température min. eau en entrée du canon' | EN: 'Min. water temperature at gun inlet'
  24 = 'CONF_Max_Temp_IN' | FR: 'Température max. eau en entrée du canon' | EN: 'Max. water temperature at gun inlet'
  25 = 'CONF_Min_Temp_OUT' | FR: 'Température min. eau en sortie du canon' | EN: 'Min. water temperature at gun outlet'
  26 = 'CONF_Max_Temp_OUT' | FR: 'Température max. eau en sortie du canon' | EN: 'Max. water temperature at gun outlet'
  27 = 'reg eau' | FR: 'Réglages température eau' | EN: 'Water temperature settings'
   = ''
END_TEXTLIST

// ---- TextLists/TextList_Config_Gaz.TcTLO
TEXTLIST TextList_Config_Gaz
  0 = 'gaz\t' | FR: 'Gaz' | EN: 'Gas'
  1 = 'definition gaz' | FR: 'Définition des gaz' | EN: 'Gas definition'
  2 = 'supervi gaz\t' | FR: 'Surveillance' | EN: 'Monitoring'
  3 = 'debit sccm' | FR: 'Tous les débits en sccm' | EN: 'All flows in sccm'
  4 = 'seuil sccm' | FR: 'Tous les seuils en sccm' | EN: 'All thresholds in sccm'
  5 = 'nom gaz nom' | FR: 'Nom du gaz\nnominal' | EN: 'Nominal\ngas name'
  6 = 'Coef' | FR: 'Coeff. de\nconversion' | EN: 'Conversion\ncoeff.'
  7 = 'debit max' | FR: 'Débit max.\ndébitmètre' | EN: 'Massflow\nmax. flow'
  8 = 'nom gaz util' | FR: 'Nom du gaz\nutilisé' | EN: 'Used gas\nname'
  9 = 'debi max gaz' | FR: 'Débit max.\ngaz' | EN: 'Gas\nmax. flow'
  11 = 'gaz1' | FR: 'Gaz 1' | EN: 'Gas 1'
  12 = 'gaz 2' | FR: 'Gaz 2' | EN: 'Gas 2'
  13 = 'gaz 3' | FR: 'Gaz 3' | EN: 'Gas 3'
  14 = 'gaz 4' | FR: 'Gaz 4' | EN: 'Gas 4'
  15 = 'gaz 5' | FR: 'Gaz 5' | EN: 'Gas 5'
  16 = 'gaz 6' | FR: 'Gaz 6' | EN: 'Gas 6'
  17 = 'gaz7' | FR: 'Gaz 7' | EN: 'Gas 7'
  18 = 'gaz8' | FR: 'Gaz 8' | EN: 'Gas 8'
  19 = 'gaz9' | FR: 'Gaz 9' | EN: 'Gas 9'
  20 = 'seuil alarme' | FR: "Seuil\nd'alarme" | EN: 'Alarm\nthreshold'
  21 = 'tps alarm' | FR: 'Temps avant\nalarme' | EN: 'Alarm\ndelay'
  22 = 'seuil défaut' | FR: 'Seuil\nde défaut' | EN: 'Fault\nthreshold'
  23 = 'tps défaut' | FR: 'Temps avant\ndéfaut' | EN: 'Fault\ndelay'
  10 = 'Purge canon' | FR: 'Purge canons à ions' | EN: 'Ions beam purge'
  24 = "Purge d'amo" | FR: "Purge d'amorcage" | EN: 'Start purge'
  25 = 'Purge stop' | FR: "Purge d'arrêt" | EN: 'Purge stop'
  26 = 'Durée' | FR: 'Durée' | EN: 'Duration'
  27 = 'Purge RAH' | FR: 'Purge atmosphère' | EN: 'Atmospheric purge'
  28 = 'Rapide' | FR: 'Rapide' | EN: 'Fast'
  29 = 'Ala surv press' | FR: 'Surveillance pression - Temps avant alarme' | EN: 'Pressure supervision - Delay before alarm'
  30 = 'def surv press' | FR: 'Surveillance pression - Temps avant défaut' | EN: 'Pressure supervision - Delay before default'
  31 = 'Gain' | FR: 'Gain' | EN: 'Amplification factor'
  32 = 'Ti' | FR: "Temps d'action intégrale" | EN: 'Integral action time'
  33 = 'Td' | FR: "Temps d'action dérivée" | EN: 'Derivative action time '
  34 = 'Ta' | FR: "Temps d'amortissment" | EN: 'Damping time'
  35 = 'Regul Gaz' | FR: 'Régulation de gaz' | EN: 'Gas regulation'
   = ''
END_TEXTLIST

// ---- TextLists/TextList_Config_IAD.TcTLO
TEXTLIST TextList_Config_IAD
  0 = 'Config IAD' | FR: 'Configuration IAD' | EN: 'IAD Configuration'
  1 = 'Seuil ala' | FR: "Seuil d'alarme" | EN: 'Alarm threshold'
  2 = 'Temps av ala' | FR: 'Temps avant alarme' | EN: 'Delay before alarm'
  3 = 'Seuil def' | FR: 'Seuil de défaut' | EN: 'Default threshold'
  4 = 'Temps av def' | FR: 'Temps avant défaut' | EN: 'Delay before fault'
  5 = 'Tension anode' | FR: "Tension d'anode" | EN: 'Anode voltage'
  6 = 'Courant anode' | FR: "Courant d'anode" | EN: 'Anode current'
  7 = 'Courant neut' | FR: 'Courant neutraliseur' | EN: 'Neutralization current'
   = ''
END_TEXTLIST

// ---- TextLists/TextList_Config_Mouvements.TcTLO
TEXTLIST TextList_Config_Mouvements
  0 = '' | FR: 'Rotation' | EN: 'Rotation'
  1 = '' | FR: 'Tilt' | EN: 'Tilt'
  2 = '' | FR: "Décalage d'origine" | EN: 'Home shift'
  3 = '' | FR: 'Erreur max. de vitesse' | EN: 'Max. speed error'
  4 = '' | FR: 'Retard défaut de surveillance vitesse' | EN: 'Speed monitoring error delay'
  5 = '' | FR: 'Limitation de couple' | EN: 'Torque limitation'
   = ''
END_TEXTLIST

// ---- TextLists/TextList_Config_Pompage.TcTLO
TEXTLIST TextList_Config_Pompage
  0 = 'Conf pomp chambre' | FR: 'Pompage chambre' | EN: 'Chamber pumping'
  1 = 'Conf pomp sas' | FR: 'Pompage sas' | EN: 'Loadlock pumping'
  2 = 'TGF' | FR: 'Seuil de détection de grosse fuite' | EN: 'Gross leak detection threshold'
  3 = 'TGF delay' | FR: 'Temps de détection grosse fuite' | EN: 'Gross leak detection time'
  4 = 'ATM' | FR: 'Seuil de pression atmosphérique' | EN: 'Atmospheric pressure threshold'
  5 = 'Surventil' | FR: 'Temps de surventilation' | EN: 'Vent overtime'
  6 = 'PPrim' | FR: 'Seuil de basculement en pompage secondaire' | EN: 'High vacuum pumping start threshold'
  7 = 'RP PPrim' | FR: 'Seuil de détection de remontée de pression' | EN: 'Pressure rise detection threshold'
  8 = 'pprim delay' | FR: 'Temps de surveillance pompage primaire' | EN: 'Rough pumping monitoring time'
  9 = 'vent delay' | FR: 'Temps de surveillance ventilation' | EN: 'Venting monitoring time'
  10 = 'prm_pr_canon_ok' | FR: "Seuil d'autorisation allumage canon à électrons" | EN: 'E-gun starting authorization threshold'
  11 = 'prm_pr_canon_ion_ok' | FR: "Seuil d'autorisation allumage canon à ions" | EN: 'Ion gun starting authorization threshold'
  12 = 'PRM_tps_att_chaud' | FR: 'Temps de thermalisation' | EN: 'Thermalisation time'
  13 = 'Conf_Temp_Min' | FR: 'Température min. groupe chaud' | EN: 'Chiller minimum temperature'
  14 = 'Conf_Temp_Max' | FR: 'Température max. groupe chaud' | EN: 'Chiller maximum temperature'
  15 = 'vanne asservie' | FR: 'Vanne asservie' | EN: 'Servovalve'
  16 = 'Estimation du temps de pompage' | FR: 'Estimation du temps de pompage' | EN: 'Estimated pumping time'
  17 = 'Pump sweep time on pump balast / intersteel pump alternation' | FR: 'Temps balayage pompe sur alternance avec pompage interjoint' | EN: 'Pump sweep time on pump balast / intersteel pump alternation'
  18 = 'Intersteel pumping time on pump balast / intersteel pump alternation' | FR: 'Temps pompage interjoint sur alternance avec balayage pompe' | EN: 'Intersteel pumping time on pump balast / intersteel pump alternation'
  19 = 'Pump balast time before pump stop' | FR: 'Temps balayage pompe avant arrêt pompe' | EN: 'Pump balast time before pump stop'
  20 = 'Primary pump balast' | FR: 'Balayage pompe primaire' | EN: 'Primary pump balast'
   = ''
END_TEXTLIST

// ---- TextLists/TextList_CryoPump.TcTLO
TEXTLIST TextList_CryoPump
  54 = 'Trame Manuelle' | FR: 'Trame Manuelle' | EN: 'Manual Frame'
  55 = 'paramètres de régénération' | FR: 'Paramètres de régénération' | EN: 'Regeneration settings'
  56 = '' | FR: 'Pompe Cryo' | EN: 'Cryo pump'
  3 = '' | FR: 'Forçage' | EN: 'Forcing'
  4 = '' | FR: 'Etat de la pompe' | EN: 'Pump Status'
  5 = '' | FR: 'Température du 1er étage (°K)' | EN: '1st stage temperature (°K)'
  6 = '' | FR: 'Température du 2ème étage (°K)' | EN: '2nd stage temperature (°K)'
  8 = 'Activé' | FR: 'Pompe activée' | EN: 'Pump activated'
  7 = 'Désactivé' | FR: 'Pompe désactivée' | EN: 'Pump disabled'
  9 = '' | FR: 'Retour' | EN: 'Back'
  10 = '' | FR: 'Temps de balayage long (min)' | EN: 'Extended purge time (min)'
  11 = '' | FR: 'Délai de redémarrage (h)' | EN: 'Delay restart (h)'
  12 = '' | FR: 'Nombre de cycles de balayage' | EN: 'Repurge cycles'
  13 = '' | FR: 'Temps de cycle du balayage (min)' | EN: 'Repurge time (min)'
  14 = '' | FR: 'Nombre de cycles de remontée en pression' | EN: 'Rate of rise cycles'
  15 = '' | FR: 'Sous pression' | EN: 'Rough to pressure'
  16 = '' | FR: "Verrouillage de la vanne d'arrêt" | EN: 'Rough Valve Interlock'
  17 = '' | FR: 'Température de démarrage (°K)' | EN: 'Start Up Temperature (°K)'
  18 = '' | FR: 'Lecture des paramètres enregistrés dans la pompe' | EN: 'Reading parameters stored in the pump'
  19 = '' | FR: 'Ecriture des paramètres dans la pompe' | EN: 'Writing parameters to the pump'
  20 = '' | FR: 'Lancer la régénération ' | EN: 'Launch regeneration '
  21 = '' | FR: 'Stopper la régénération ' | EN: 'Stop regeneration '
  22 = '' | FR: 'Commande :' | EN: 'Command :'
  23 = '' | FR: 'Réponse :' | EN: 'Response :'
  24 = '' | FR: 'Envoie Trame ' | EN: 'Send Frame'
  25 = '' | FR: 'Pompe Cryo On-Board' | EN: 'CryoPump On-Board'
  26 = '' | FR: 'ÉCHAUFFEMENT' | EN: 'WARM-UP'
  27 = '' | FR: 'DÉFAILLANCE DU GAZ DE PURGE' | EN: 'PURGE GAS FAILURE'
  28 = '' | FR: 'Balayage long' | EN: 'Extended purge'
  29 = '' | FR: 'Pression de pompage primaire (μ)' | EN: 'Rough to base pressure (μ)'
  30 = '' | FR: 'Remontée en pression ROR (μ/min)' | EN: 'Rate of rise ROR (μ/min)'
  31 = '' | FR: 'REFROIDISSEMENT' | EN: 'COOLDOWN'
  32 = '' | FR: 'DÉLAI DE REDÉMARRAGE' | EN: 'DELAY RESTART'
  33 = '' | FR: 'DÉLAI DE DÉMARRAGE' | EN: 'DELAY START'
  34 = '' | FR: 'RÉGÉNÉRATION TERMINÉE' | EN: 'REGEN COMPLETED'
  35 = '' | FR: 'RÉGÉNÉRATION ARRÊTÉE' | EN: 'REGEN ABORTED'
  36 = '' | FR: "Retour aux paramètres d'usine" | EN: 'Return to factory settings'
  38 = '' | FR: 'Ouverte' | EN: 'Open'
  37 = '' | FR: 'Fermé' | EN: 'Close'
  39 = '' | FR: 'Etat de la vanne primaire' | EN: 'Rough Valve Status'
  40 = '' | FR: 'Etat de la vanne de balayage' | EN: 'Purge Valve Status'
  41 = '' | FR: 'Vanne primaire' | EN: 'Rough Valve'
  42 = '' | FR: 'Vanne de balayage' | EN: 'Purge Valve'
  43 = '' | FR: 'Etapes de la régénération en cours :' | EN: 'Stages of regeneration in progress :'
  44 = '' | FR: 'Cryo éteinte' | EN: 'Cryo Off'
  45 = '' | FR: 'Rétablissement après coupure' | EN: 'Power Fail Recovery'
  46 = '' | FR: 'Informations de la pompe' | EN: 'Pump Infos'
  47 = '' | FR: 'Numéro de série de la pompe' | EN: 'Pump Serial Number'
  48 = '' | FR: 'Nombre de cycles de régénération completés' | EN: 'Number of complete regeneration'
  49 = '' | FR: 'Temps depuis la dernière régénération (h)' | EN: 'Time since last regeneration (h)'
  50 = '' | FR: 'Niveau de révision du logiciel' | EN: 'Software revision level'
  51 = '' | FR: 'Temps de fonctionnement de la pompe (h)' | EN: 'Pump operating time (h)'
  52 = '' | FR: 'Réinitialiser ' | EN: 'RESET'
  53 = '' | FR: 'Pression (μ)' | EN: 'Pressure (μ)'
  0 = '' | FR: 'OFF' | EN: 'OFF'
  1 = '' | FR: 'ON' | EN: 'ON'
  2 = '' | FR: 'COOL' | EN: 'COOL'
  57 = '' | FR: 'Délai de démarrage (h)' | EN: 'Delay start (h)'
  58 = '' | FR: "TEMPS D'ÉCHAUFFEMENT" | EN: 'WARMUP TIMEOUT'
  59 = '' | FR: 'AUCUNE ERREUR' | EN: 'NO ERROR'
  60 = '' | FR: 'DÉLAI DE REFROIDISSEMENT' | EN: 'COOLDOWN TIMEOUT'
  61 = '' | FR: 'ERREUR DANS LE ROR' | EN: 'ERROR IN ROR'
  62 = '' | FR: 'LA LIMITE DE CYCLES ROR A ÉTÉ ATTEINTE' | EN: 'ROR CYCLE LIMIT WAS REACHED'
  63 = '' | FR: 'ARRÊT MANUEL' | EN: 'MANUAL ABORT'
  64 = '' | FR: "DÉLAI D'ATTENTE DE LA VANNE PRIMAIRE" | EN: 'ROUGH VALVE TIMEOUT'
  65 = '' | FR: 'BOGUE DU SYSTÈME' | EN: 'SYSTEM BUG'
  66 = '' | FR: 'Numero du relais :' | EN: 'Relay number :'
  67 = '' | FR: 'Commande du paramètre :' | EN: 'Settings command :'
  68 = '' | FR: 'Valeur :' | EN: 'Value :'
  69 = '' | FR: 'Appliquer ces paramètres' | EN: 'Apply this settings'
  70 = '' | FR: 'Température du 1er étage' | EN: '1st stage temperature'
  71 = '' | FR: 'Température de 2ème étage' | EN: '2nd stage temperature'
  72 = '' | FR: 'Pression Cryo TC' | EN: 'Cryo TC pressure'
  73 = '' | FR: 'Pression TC auxiliaire' | EN: 'Aux TC pressure'
  74 = '' | FR: "Délai d'attente (passage ON/OFF)" | EN: 'Time delay (switch ON/OFF)'
  75 = '' | FR: 'Fonction manuelle = ON' | EN: 'Manual Function = ON'
  76 = '' | FR: 'Fonction manuelle = OFF' | EN: 'Manual Function = OFF'
  77 = '' | FR: "Suivi de l'état de régénération" | EN: 'Regen track'
  78 = '' | FR: "Suivi de l'état de vanne primaire" | EN: 'Rough valve track'
  79 = '' | FR: "Suivi de l'état de la pompe cryo" | EN: 'Cryopump track'
  80 = '' | FR: 'Paramétrages des relais' | EN: 'Relay settings'
  81 = '' | FR: 'Mode manuel' | EN: 'Manual mode'
  82 = '' | FR: 'Mode automatique' | EN: 'Automatic mode'
  84 = '' | FR: 'Relais actif (ON)' | EN: 'Enable relay (ON)'
  83 = '' | FR: 'Relais inactif (OFF)' | EN: 'Disable relay (OFF)'
  85 = '' | FR: 'Restaure les paramètres automatiques' | EN: 'Restores automatic settings'
  86 = '' | FR: 'Cycle de rebalayage' | EN: 'Repurge cycle'
  1000 = '' | FR: 'Pas de données' | EN: 'No data'
  87 = '' | FR: 'Informations supplémentaires' | EN: 'Further information'
  88 = '' | FR: 'Lecture ' | EN: 'Read'
  89 = '' | FR: 'Attention !' | EN: 'Warning !'
  90 = '' | FR: 'Cette action peut altérer le bon fonctionnement de la machine. Voulez-vous continuer ?' | EN: "This action may affect the machine's operation. Do you want to continue?"
  91 = '' | FR: "Êtes-vous sûr de retourner aux paramètres d'usine ?" | EN: 'Are you sure you want to return to factory settings ?'
  92 = '' | FR: 'Confirmer' | EN: 'Confirm'
  93 = '' | FR: 'Annuler' | EN: 'Cancel'
  94 = '' | FR: 'Etats' | EN: 'States'
  95 = '' | FR: 'Fermé' | EN: 'Closed'
  96 = '' | FR: 'Régulation de la température du 1er étage' | EN: '1st floor temperature control'
  97 = '' | FR: 'maintenance alliance concept' | EN: 'alliance concept maintenance'
  98 = '' | FR: 'Configuration de la pompe cryo' | EN: 'Cryo pump settings'
   = ''
END_TEXTLIST

// ---- TextLists/TextList_Cryo_Relays_Parameters.TcTLO
TEXTLIST TextList_Cryo_Relays_Parameters
  0 = '' | FR: 'Régler le seuil inférieur du 1er étage (deg Kelvin)' | EN: 'Set first stage LL (deg Kelvin)'
  1 = '' | FR: 'Régler le seuil supérieur du 1er étage (deg Kelvin)' | EN: 'Set first stage UL (deg Kelvin)'
  2 = '' | FR: 'Régler le seuil inférieur du 2ème étage (deg Kelvin)' | EN: 'Set second stage LL (deg Kelvin)'
  3 = '' | FR: 'Régler le seuil supérieur du 2ème étage (deg Kelvin)' | EN: 'Set second stage UL (deg Kelvin)'
  4 = '' | FR: 'Régler la pression inférieure du thermocouple de la cryo (microns)' | EN: 'Set Pump TC LL (microns)'
  5 = '' | FR: 'Régler la pression supérieure du thermocouple de la cryo (microns)' | EN: 'Set Pump TC UL (microns)'
  6 = '' | FR: 'Régler la pression inférieure du thermocouple auxiliaire (microns)' | EN: 'Set AUX TC LL (microns)'
  7 = '' | FR: 'Régler la pression supérieure du thermocouple auxiliaire (microns)' | EN: 'Set AUX TC UL (microns)'
  8 = '' | FR: 'Régler le temps du relais (0-9999 secondes)' | EN: 'Set time relay (0-9999 seconds)'
  10 = '' | FR: 'Activation inconditionnelle' | EN: 'Set unconditional ON'
  11 = '' | FR: 'Désactivation inconditionnelle' | EN: 'Set unconditional OFF'
  12 = '' | FR: "Régler le suivi de l'état de régénération" | EN: 'Set as REGEN status tracking relay'
  13 = '' | FR: "Régler le suivi de l'état de vanne primaire" | EN: 'Set as rough valve tracking relay'
  15 = '' | FR: "Régler le suivi de l'état de la pompe cryo" | EN: 'Set as pump motor ON/OFF status tracking relay'
  9 = '' | FR: '-' | EN: '-'
  14 = '' | FR: '-' | EN: '-'
   = ''
END_TEXTLIST

// ---- TextLists/TextList_EcoMode.TcTLO
TEXTLIST TextList_EcoMode
  0 = 'Activation Eco-veille' | FR: 'Activation Eco-veille' | EN: 'Eco-sleep activation'
  1 = 'Temps inav' | FR: "Temps d'inactivité avant Eco-veille" | EN: 'Inactivity time before eco-sleep'
  2 = 'Process deep eco-sleep' | FR: 'Procédé Eco-veille profond' | EN: 'Deep eco-sleep process'
  3 = 'Record' | FR: 'Enregistrement' | EN: 'Record'
  4 = 'Select' | FR: '...' | EN: '...'
  5 = 'Canon actif' | FR: 'Evap. active' | EN: 'Evap. on'
  6 = 'On/Off' | FR: 'Activation/Désactivation' | EN: 'On/Off'
  7 = 'Evap On/Off' | FR: 'Activation/Désactivation Evap.' | EN: 'Evap. On/Off'
  8 = 'Eco Mode' | FR: 'Eco-veille' | EN: 'Eco-sleep'
  9 = 'Config' | FR: 'Configuration' | EN: 'Configuration'
  10 = 'Eco Mode actif' | FR: 'Eco-veille actif' | EN: 'Eco-sleep On'
  11 = 'Inactivité' | FR: 'Inactivité :' | EN: 'Inactivity :'
  12 = " Lancement du procédé eco-veille profond à l'issue de la production" | FR: " Lancement du procédé Eco-veille profond à l'issue de la production" | EN: 'Start the deep eco-sleep process at the end of the production'
   = ''
END_TEXTLIST

// ---- TextLists/TextList_Effluvage.TcTLO
TEXTLIST TextList_Effluvage
  0 = ''
  1 = 'EFFLUVAGE' | FR: 'EFFLUVAGE' | EN: 'GLOW DISCHARGE'
  2 = 'Courant' | FR: 'Courant' | EN: 'Current'
  3 = 'time' | FR: 'Temps' | EN: 'Timer'
  4 = 'PT' | FR: 'Temps écoulé' | EN: 'Passed time'
  5 = 'Tension attendue' | FR: 'Tension attendue' | EN: 'Expected voltage'
  6 = ''
  7 = ''
   = ''
END_TEXTLIST

// ---- TextLists/TextList_Evap.TcTLO
TEXTLIST TextList_Evap
  0 = '' | FR: 'Creuset' | EN: 'Crucible'
  1 = '' | FR: 'Balayage' | EN: 'Sweeping'
  2 = '' | FR: 'Courant' | EN: 'Current'
  3 = '' | FR: 'Haute Tension' | EN: 'High Voltage'
  4 = '' | FR: 'Consigne' | EN: 'Setpoint'
  5 = 'Etat' | FR: 'Etat' | EN: 'State'
   = ''
END_TEXTLIST

// ---- TextLists/TextList_Gaz.TcTLO
TEXTLIST TextList_Gaz
  0 = 'select' | FR: 'Sélectionner' | EN: 'Select'
  1 = 'ouvert' | FR: 'Ouverte' | EN: 'Opened'
  2 = 'fermé' | FR: 'Fermée' | EN: 'Closed'
  11 = 'ligne 1' | FR: 'Ligne de gaz 1' | EN: 'Gas line 1'
  12 = 'ligne 2' | FR: 'Ligne de gaz 2' | EN: 'Gas line 2'
  13 = 'ligne 3' | FR: 'Ligne de gaz 3' | EN: 'Gas line 3'
  14 = 'ligne 4' | FR: 'Ligne de gaz 4' | EN: 'Gas line 4'
  3 = 'debit' | FR: 'Débit (sccm)' | EN: 'Flow (sccm)'
  15 = 'Consigne pos' | FR: 'Consigne de position (%)' | EN: 'Position setpoint (%)'
  16 = 'Consigne pres' | FR: 'Consigne de pression (mbar)' | EN: 'Pressure setpoint (mbar)'
  17 = 'Press min' | FR: 'Pression min. (mbar)' | EN: 'Min. pressure (mbar)'
  18 = 'Press max' | FR: 'Pression max. (mbar)' | EN: 'Max. pressure (mbar)'
  19 = 'Temps stab' | FR: 'Temps de stab.' | EN: 'Stab. time'
   = ''
END_TEXTLIST

// ---- TextLists/TextList_IAD.TcTLO
TEXTLIST TextList_IAD
  0 = '' | FR: "Tension d'anode" | EN: 'Anode voltage'
  1 = '' | FR: "Courant d'anode" | EN: 'Anode current'
  2 = '' | FR: 'Courant neutraliseur' | EN: 'Neutralization current'
  3 = '' | FR: 'Pourcentage gaz 1' | EN: 'Gas 1 pourcent'
  4 = '' | FR: 'Pourcentage gaz 2' | EN: 'Gas 2 pourcent'
  5 = '' | FR: 'Durée' | EN: 'Time'
  6 = '' | FR: 'Temps écoulé' | EN: 'Elapsed time'
  7 = '' | FR: "Débit d'amorcage gaz 1" | EN: 'Starting gas 1 flow'
  8 = '' | FR: "Débit d'amorcage gaz 2" | EN: 'Starting gas 2 flow'
  9 = '' | FR: "Débit d'amorcage gaz  HCES" | EN: 'Starting gas HCES flow'
  10 = '' | FR: 'Canon à ions' | EN: 'Ions gun'
  11 = '' | FR: 'Temps' | EN: 'Time'
  12 = '' | FR: 'Temps écoulé' | EN: 'Time elapsed'
   = ''
END_TEXTLIST

// ---- TextLists/TextList_IC6.TcTLO
TEXTLIST TextList_IC6
  0 = 'Rate' | FR: 'Vitesse (Å/s)' | EN: 'Rate (Å/s)'
  1 = 'Thickness' | FR: 'Epaisseur (kÅ)' | EN: 'Thickness (kÅ)'
  2 = 'Détails' | FR: 'Détails...' | EN: 'Details...'
  3 = 'power' | FR: 'Puissance (%)' | EN: 'Power (%)'
  4 = 'Commandes' | FR: ' Commandes' | EN: ' Commands'
  5 = 'start' | FR: 'START' | EN: 'START'
  6 = 'stop' | FR: 'STOP' | EN: 'STOP'
  7 = 'ZERO' | FR: 'ZERO' | EN: 'ZERO'
  8 = 'RESET' | FR: 'RESET' | EN: 'RESET'
  9 = 'etat quartz' | FR: ' Etat des quartz' | EN: ' Crystals state'
  10 = 'fail' | FR: 'FAIL' | EN: 'FAIL'
  11 = 'channel' | FR: 'Canal actif :' | EN: 'Active channel:'
  12 = 'Fréquence' | FR: 'Fréquence' | EN: 'Frequency'
  13 = '% utilisé' | FR: '% utilisé' | EN: 'Life used'
  14 = 'Etat quartz' | FR: 'Etat quartz' | EN: 'Crystal quartz'
   = ''
END_TEXTLIST

// ---- TextLists/TextList_Infos.TcTLO
TEXTLIST TextList_Infos
  0 = 'Langue' | FR: 'Langue' | EN: 'Language'
  1 = 'Id' | FR: 'Affaire :' | EN: 'Id:'
  2 = 'Auteur' | FR: 'Auteur :' | EN: 'Author:'
  3 = 'version' | FR: 'Version :' | EN: 'Release:'
  4 = 'date' | FR: 'Date :' | EN: 'Date:'
  5 = 'num' | FR: 'N° de série :' | EN: 'Serial number:'
  6 = 'type' | FR: 'Modèle :' | EN: 'Type:'
   = ''
END_TEXTLIST

// ---- TextLists/TextList_Moteurs.TcTLO
TEXTLIST TextList_Moteurs
  0 = '' | FR: 'Reset Moteur' | EN: 'Motor Reset'
  1 = '' | FR: 'Reset Position' | EN: 'Position Reset'
  2 = '' | FR: 'Dévalidation' | EN: 'Devalidation'
  3 = '' | FR: 'Compteur de\nbalayages' | EN: 'Sweepings\nCounter'
  4 = '' | FR: 'Aller en position de transfert' | EN: 'Go to transfer position'
  5 = '' | FR: 'Position\nBasse' | EN: 'Low\nPosition'
  6 = '' | FR: 'Position\nHaute' | EN: 'High\nPosition'
  7 = '' | FR: 'Vitesse' | EN: 'Speed'
  8 = '' | FR: 'Poste' | EN: 'Station'
  9 = '' | FR: 'Distance' | EN: 'Distance'
  10 = '' | FR: 'De' | EN: 'From'
  11 = '' | FR: 'Réf.' | EN: 'Homed'
  12 = '' | FR: 'Position' | EN: 'Position'
  13 = '' | FR: 'Poste sélectionné' | EN: 'Selected station'
  14 = '' | FR: 'Référence sélectionnée' | EN: 'Selected reference'
  15 = '' | FR: 'Consignes' | EN: 'Setpoints'
  16 = '' | FR: 'Amplitude balayage' | EN: 'Sweeping amplitude'
  17 = '' | FR: 'Accélération' | EN: 'Acceleration'
  18 = '' | FR: 'Décélération' | EN: 'Deceleration'
  19 = '' | FR: 'Avec prise\nde référence' | EN: 'With\nHoming'
  20 = '' | FR: 'Sans prise\nde référence' | EN: 'Without\nHoming'
  21 = '' | FR: 'Départ centré' | EN: 'Centered start'
  22 = '' | FR: 'Départ déporté' | EN: 'Deported start'
   = ''
END_TEXTLIST

// ---- TextLists/TextList_Navigation.TcTLO
TEXTLIST TextList_Navigation
  0 = 'Syn pomp' | FR: 'Synoptique\nPompage' | EN: 'Pumping\nSynoptic'
  1 = 'Syn proc' | FR: 'Synoptique\nProcédé' | EN: 'Process\nSynoptic'
  2 = 'SA'
  3 = 'Conf pomp' | FR: 'Pompage' | EN: 'Pumping'
  4 = 'Conf evap' | FR: 'Evaporation' | EN: 'Evaporation'
  5 = 'Conf mvts' | FR: 'Mouvements' | EN: 'Movements'
  6 = 'sa pomp ch' | FR: 'Pompage chambre' | EN: 'Chamber pumping'
  7 = 'sa pomp sas' | FR: 'Pompage sas' | EN: 'Loadlock pumping'
  8 = 'Conf gaz\t' | FR: 'Gaz' | EN: 'Gas'
  9 = 'Conf IAD' | FR: 'IAD' | EN: 'IAD'
  10 = 'Conf Chauf' | FR: 'Chauffage' | EN: 'Heating'
  11 = 'Effluvage' | FR: 'Effluvage' | EN: 'Glow discharge'
  12 = 'Conf Serv' | FR: 'Servitudes' | EN: 'Easements'
  13 = 'Cryo' | FR: 'Cryo' | EN: 'Cryo'
   = ''
END_TEXTLIST

// ---- TextLists/TextList_Orders.TcTLO
TEXTLIST TextList_Orders
  0 = 'open' | FR: 'Ouvrir' | EN: 'Open'
  1 = 'close' | FR: 'Fermer' | EN: 'Close'
  2 = 'Clampage' | FR: 'Clampage' | EN: 'Clamping'
  3 = 'Déclampage' | FR: 'Déclampage' | EN: 'Unclamping'
   = ''
END_TEXTLIST

// ---- TextLists/TextList_Pompage.TcTLO
TEXTLIST TextList_Pompage
  0 = 'Pomp inter' | FR: 'Pompage interjoints' | EN: 'Inter ring pumping'
  1 = 'Confirm regen' | FR: 'Confirmer régénération ?' | EN: 'Confirm regeneration ?'
   = ''
END_TEXTLIST

// ---- TextLists/TextList_Position_Canne.TcTLO
TEXTLIST TextList_Position_Canne
  0 = 'sas' | FR: 'Sas (0)' | EN: 'Loadlock (0)'
  1 = 'egun1' | FR: 'Canon 1' | EN: 'E-gun 1'
  2 = 'evap' | FR: 'Source Joule' | EN: 'Thermal source'
  3 = 'egun2' | FR: 'Canon 2' | EN: 'E-gun 2'
  255 = 'undefined' | FR: 'Indéfinie' | EN: 'Undefined'
   = ''
END_TEXTLIST

// ---- TextLists/TextList_Process.TcTLO
TEXTLIST TextList_Process
  0 = 'Selec proc' | FR: 'Procédé sélectionné :' | EN: 'Selected process:'
  1 = 'step' | FR: 'Etape en cours :' | EN: 'Step in progress:'
  2 = 'layer' | FR: 'Couche :' | EN: 'Layer:'
  3 = 'start' | FR: 'Marche\nProduction' | EN: 'Start\nProduction'
  4 = 'stop' | FR: 'Arrêt\nProduction' | EN: 'Stop\nProduction'
  5 = 'inter' | FR: 'Interruption\nProduction' | EN: 'Break\nProduction'
  6 = 'resume' | FR: 'Reprise\nProduction' | EN: 'Resume\nProduction'
  7 = 'process name' | FR: 'Nom procédé' | EN: 'Process name'
  8 = 'etape' | FR: 'Etape' | EN: 'Step'
  9 = 'type etape' | FR: 'Type étape' | EN: 'Step type'
  10 = 'tps effluvage' | FR: 'Durée effluvage' | EN: 'Glow disch. time'
  11 = 'couche' | FR: 'Couche' | EN: 'Layer'
  12 = 'détails' | FR: 'Détails' | EN: 'Details'
  13 = 'boucle' | FR: 'Boucle' | EN: 'Loop'
  14 = 'first' | FR: 'Départ' | EN: 'First'
  15 = 'fin' | FR: 'Fin' | EN: 'Last'
  16 = 'seg' | FR: 'Segment' | EN: 'Segment'
  17 = 'tps seg' | FR: 'Temps segment' | EN: 'Segment time'
  18 = 'tps couche' | FR: 'Temps couche' | EN: 'Layer time'
  19 = 'next layer' | FR: 'Couche suivante' | EN: 'Next layer'
  20 = 'break' | FR: 'Interruption' | EN: 'Break'
  21 = 'resume' | FR: 'Reprise' | EN: 'Resume'
  22 = 'arrêt' | FR: 'Arrêt procédé' | EN: 'Process stop'
  23 = 'next step' | FR: 'Etape suivante' | EN: 'Next step'
  24 = 'Temps purge' | FR: 'Temps purge' | EN: 'Purge time'
  25 = 'Temps etching' | FR: 'Temps décapage' | EN: 'Etching time'
  26 = 'Rechargement' | FR: 'Rechargement' | EN: 'Reload'
   = ''
END_TEXTLIST

// ---- TextLists/TextList_SA_Operations.TcTLO
TEXTLIST TextList_SA_Operations
  0 = 'Pompage' | FR: 'Pompage' | EN: 'Pumping'
  1 = 'Marche pompe' | FR: 'Marche\nPompes' | EN: 'Start\nPumps'
  2 = 'Arret pompe' | FR: 'Arrêt\nPompes' | EN: 'Stop\nPumps'
  3 = 'Isol' | FR: 'Isolement' | EN: 'Standby'
  4 = 'Vent' | FR: 'Ventilation' | EN: 'Venting'
  5 = 'Marche' | FR: 'Marche' | EN: 'Start'
  6 = 'Validation' | FR: 'Validation' | EN: 'Validation'
  7 = 'Arrêt' | FR: 'Arrêt' | EN: 'Stop'
  8 = 'Position' | FR: 'Positionnement' | EN: 'Positioning'
  9 = 'Initialisation' | FR: 'Repli' | EN: 'Folding'
  10 = 'cooling' | FR: "Refroidissement\nd'urgence" | EN: 'Emergency\nCooling'
  11 = 'pomp proc' | FR: 'Pompage\nProcédé' | EN: 'Process\nPumping'
  12 = 'on gaz' | FR: 'Mise en\ngaz' | EN: 'Start\ngas'
  13 = 'off gaz' | FR: 'Arrêt\ngaz' | EN: 'Stop\ngas'
  14 = 'rampee' | FR: 'Rampe\ngaz' | EN: 'Gas\nramp'
  15 = 'rotation' | FR: 'Rotation' | EN: 'Rotation'
  16 = 'Bal' | FR: 'Balayage' | EN: 'Sweeping'
  17 = 'regen' | FR: 'Régénération\nCryo' | EN: 'Cryo\nRegeneration'
  18 = 'charg' | FR: 'Chargement\nChambre' | EN: 'Chamber\nLoading'
  19 = 'decharg' | FR: 'Déchargement\nChambre' | EN: 'Chamber\nUnloading'
  20 = 'Init' | FR: 'Initialisation' | EN: 'Initialization'
  21 = 'Scan quartz' | FR: 'Scan quartz' | EN: 'Scan crystal'
  22 = 'Positionnement quartz' | FR: 'Positionnement quartz' | EN: 'Position crystal'
  23 = 'Position' | FR: 'Position' | EN: 'Position'
  24 = 'marche ch' | FR: 'Marche\nchauffage' | EN: 'Start\nheating'
  25 = 'arret ch' | FR: 'Arrêt\nchauffage' | EN: 'Stop\nheating'
  26 = 'Marche decap' | FR: 'Marche décapage' | EN: 'Start ion etching'
  27 = 'Stop decap' | FR: 'Arrêt décapage' | EN: 'Stop ion etching'
  28 = 'Pompage prim' | FR: 'Pompage\nprimaire' | EN: 'Primary\npumping'
  29 = 'Marche' | FR: 'Marche' | EN: 'Start'
   = ''
END_TEXTLIST

// ---- TextLists/TextList_Servitudes.TcTLO
TEXTLIST TextList_Servitudes
  0 = 'Groupe froid' | FR: 'Circulateur Chaud / Froid' | EN: 'Hot / Cold circulator'
  4 = '' | FR: "Tempéraure maximale de l'eau en sortie avant défaut" | EN: 'Maximum temperature for output water before fault'
  3 = '' | FR: "Tempéraure minimale de l'eau en sortie avant défaut" | EN: 'Minimum temperature for output water before fault'
  2 = '' | FR: "Débit maximal de l'eau en sortie avant défaut" | EN: 'Maximum flow for output water before fault'
  1 = '' | FR: "Débit minimal de l'eau en sortie avant défaut" | EN: 'Minimum flow for output water before fault'
  5 = '' | FR: "Tempéraure maximale de l'eau en sortie avant alarme" | EN: 'Maximum temperature for output water before warning'
   = ''
END_TEXTLIST

// ---- TextLists/TextList_STATE_Mode_Marche.TcTLO
TEXTLIST TextList_STATE_Mode_Marche
  0 = '0 - PLC Off' | FR: "0 - Automate à l'arrêt" | EN: '0 - PLC Off'
  1 = '1 - PLC Starting' | FR: '1 - Démarrage automate' | EN: '1 - PLC starting'
  2 = '2 - Waiting for\nmachine supply' | FR: '2 - Attente\nalimentation machine' | EN: '2 - Waiting for machine supply'
  3 = '3 - Machine stopped' | FR: "3 - Machine à l'arrêt" | EN: '3 - Machine stopped'
  4 = '4 - Waiting for operating\nmode selection...' | FR: '4 - Attente sélection\nmode de marche...' | EN: '4 - Wait for operating mode selection...'
  5 = '5 - Machine initialization...' | FR: '5 - Initialisation machine' | EN: '5 - Machine initialization'
  6 = '6 - Automatic mode' | FR: '6 - Mode automatique' | EN: '6 - Automatic mode'
  7 = '7 - Production preparation' | FR: '7 - Préparation production' | EN: '7 - Production preparation'
  8 = '8 - Production' | FR: '8 - Production en cours...' | EN: '8 - Production in progress...'
  9 = '9 - Production stopped' | FR: '9 - Production stoppée' | EN: '9 - Production stopped'
  10 = '10 - Manual mode' | FR: '10 - Mode manuel' | EN: '10 - Manual mode'
  11 = '11 - Fin de production' | FR: '11 - Fin de production' | EN: '11 - End of production'
  12 = '12 - Interruption de production' | FR: '12 - Interruption de production' | EN: '12 - Production interruption'
  13 = '13 - En attente de reprise' | FR: '13 - En attente de reprise' | EN: '13 - Waiting for resume'
  20 = '20 - Lancement Eco' | FR: '20 - Lancement Eco Mode' | EN: '20 - Eco Mode starting'
  21 = '21 - Eco Mode' | FR: '21 - Eco Mode' | EN: '21 - Eco Mode'
  22 = '22 - Lancement procédé\neco-veille profond' | FR: '22 - Lancement procédé\neco-veille profond' | EN: '22 - Deep eco-sleep process starting'
  23 = '23 - Lancement procédé\neco-veille profond' | FR: '23 - Lancement procédé\neco-veille profond' | EN: '23 - Deep eco-sleep process starting'
  24 = '24 - Procédé eco-veille\nprofond en cours' | FR: '24 - Procédé eco-veille\nprofond en cours' | EN: '24 - Deep eco-sleep process running'
  25 = '25 - Arrêt procédé\neco-veille profond' | FR: '25 - Arrêt procédé\neco-veille profond' | EN: '25 - Deep eco-sleep process end'
  26 = '26 - Procédé eco-veille\nprofond en défaut' | FR: '26 - Procédé eco-veille\nprofond en défaut' | EN: '26 - Deep eco-sleep process in fault'
  27 = '27 - Attente sortie de veille\nappareils' | FR: '27 - Attente sortie de veille\nappareils' | EN: '27 - Waiting for devices wakes up'
   = ''
END_TEXTLIST

// ---- TextLists/TextList_Test_RP.TcTLO
TEXTLIST TextList_Test_RP
  0 = 'tes trp' | FR: 'Test de remontée de pression' | EN: 'Pressure rise test'
  1 = 'init' | FR: 'Pression initiale' | EN: 'Initial pressure'
  2 = 'tps isol' | FR: "Durée d'isolement" | EN: 'Standby duration'
  3 = 'volume' | FR: 'Volume' | EN: 'Volume'
  4 = 'tps ecoul' | FR: 'Durée écoulée' | EN: 'Elapsed time'
  5 = 'result' | FR: 'Résultat :' | EN: 'Result:'
  6 = 'arret' | FR: 'Arrêt' | EN: 'Stop'
   = ''
END_TEXTLIST

// ---- TextLists/TextList_Type_Etape.TcTLO
TEXTLIST TextList_Type_Etape
  0 = 'Aucun' | FR: 'Aucun' | EN: 'None'
  1 = '' | FR: 'Pompage chambre' | EN: 'Chamber pumping'
  2 = '' | FR: 'Isolement chambre' | EN: 'Chamber standby'
  3 = '' | FR: 'Marche pompes chambre' | EN: 'Chamber pumps start'
  4 = '' | FR: 'Arrêt pompes chambre' | EN: 'Chamber pumps stop'
  5 = '' | FR: 'Régénération pompe cryogénique' | EN: 'Cryo Pump regeneration'
  6 = '' | FR: 'Ventilation chambre' | EN: 'Chamber venting'
  7 = '' | FR: "Point d'arrêt" | EN: 'Break point'
  8 = '' | FR: 'Evaporation' | EN: 'Evaporation'
  9 = '' | FR: 'Synchronisation horaire' | EN: 'Time synchronization'
  10 = '' | FR: 'Temporisation' | EN: 'Timer'
  11 = '' | FR: 'Rotation PS' | EN: 'SH Rotation'
  12 = '' | FR: 'Arrêt rotation PS' | EN: 'SH Stop Rotation'
  13 = '' | FR: 'Effluvage' | EN: 'Glow discharge'
  14 = '' | FR: 'Test de remontée de pression' | EN: 'Pressure rise test'
  15 = '' | FR: 'Arrêt procédé' | EN: 'Stopping process'
  16 = '' | FR: 'Boucle/Saut' | EN: 'Loop/Skip'
  17 = '' | FR: 'Lancement Eco-veille' | EN: 'Start Eco-sleep'
  18 = '' | FR: 'Arrêt Eco-veille' | EN: 'Stop Eco-sleep'
  19 = '' | FR: 'Régénération partielle cryo' | EN: 'Cryo pump partial regeneration'
   = ''
END_TEXTLIST

// ---- TextLists/TextList_Type_Moteur.TcTLO
TEXTLIST TextList_Type_Moteur
  0 = '' | FR: 'NU' | EN: 'NU'
  1 = '' | FR: 'Rotation PS' | EN: 'SH Rotation'
  2 = '' | FR: 'Translation PS' | EN: 'SH Translation'
  3 = '' | FR: 'Ascenseur' | EN: 'Stacker'
  4 = '' | FR: 'Rotation' | EN: 'Rotation'
  5 = '' | FR: 'Déploiement' | EN: 'Deployement'
  6 = '' | FR: 'Translation' | EN: 'Translation'
  7 = '' | FR: 'Porte Substrat' | EN: 'Substrate Holder'
  8 = '' | FR: 'Caches' | EN: 'Shutters'
  9 = '' | FR: 'Satellisation' | EN: 'Satellization'
  10 = '' | FR: 'Tilt Porte Substrat' | EN: 'Substrate holder Tilt'
   = ''
END_TEXTLIST

// ---- TextLists/TextList_Users_Menu.TcTLO
TEXTLIST TextList_Users_Menu
  1 = 'Gestion des utilisateurs\n' | FR: 'Gestion des utilisateurs' | EN: 'User management'
  2 = 'Identifiant' | FR: 'Identifiant' | EN: 'Login'
  17 = 'Save on disk' | FR: "Les groupes et utilisateurs\nvont être sauvegardés sur le disque.\nL'ancienne sauvegarde sera supprimée.\nConfirmer?" | EN: 'Users and groups will be \nsaved on disk. \nLast backup will be deleted. \nConfirm?'
  3 = 'Déconnexion' | FR: 'Confimez vous la déconnexion?' | EN: 'Confirm disconnection?'
  4 = 'Identification' | FR: 'Identification' | EN: 'Identification'
  5 = 'Login' | FR: 'Identifiant' | EN: 'Login'
  6 = 'Password' | FR: 'Mot de passe' | EN: 'Password'
  19 = 'Confirm supp groupe' | FR: 'Confirmer la suppression du groupe?' | EN: 'Confirm the group deletion?'
  18 = 'Confirm supp user' | FR: "Confirmer la suppression de l'utilisateur?" | EN: 'Confirm the user deletion?'
  21 = 'Confirm pwd' | FR: 'Confimation du mot de passe' | EN: 'Password confirmation'
  30 = 'Temps av deco' | FR: 'Temps avant déconnexion automatique :' | EN: 'Time before automatic logout:'
  31 = 'Deco auto utilisee' | FR: 'Utilisation de la déconnexion automatique :' | EN: 'Automatic logout used:'
  7 = 'user actu' | FR: 'Utilisateur actuel' | EN: 'Current user'
  8 = 'group actu' | FR: 'Groupe' | EN: 'Group'
  9 = 'Connexion' | FR: 'Connexion' | EN: 'Connection'
  10 = 'Déconnexion' | FR: 'Déconnexion' | EN: 'Disconnection'
  11 = 'droits par défaut' | FR: 'Droits\npar défaut' | EN: 'Rights\nby default'
  12 = 'Users' | FR: 'Utilisateurs' | EN: 'Users'
  13 = 'Groups' | FR: 'Groupes' | EN: 'Groups'
  14 = 'Charger' | FR: 'Charger' | EN: 'Load'
  15 = 'Sauvegarder' | FR: 'Sauvegarder' | EN: 'Save'
  16 = 'Options' | FR: 'Options' | EN: 'Options'
  20 = 'laod from disk' | FR: 'Les groupes et utilisateurs\nvont être restaurés depuis le disque\nLes groupes et utilisateurs actuels \nvont être écrasés. Confirmer?' | EN: 'Users and groups will be \nrestored from disk. \nCurrent groups and users will be deleted. \nConfirm?'
   = ''
END_TEXTLIST

// ---- TextLists/TextList_Util_Defaut.TcTLO
TEXTLIST TextList_Util_Defaut
  1 = 'Défaut' | FR: 'Droits par défaut' | EN: 'Rights by default'
   = ''
END_TEXTLIST

// ---- TextLists/TextList_Util_Group.TcTLO
TEXTLIST TextList_Util_Group
  1 = 'Liste des groupes' | FR: 'Liste des groupes' | EN: 'Group list'
  3 = 'Edition procédés' | FR: 'Edition procédés' | EN: 'Process edition'
  4 = 'Maintenance' | FR: 'Maintenance' | EN: 'Maintenance'
  5 = 'Administrateur' | FR: 'Administrateur' | EN: 'Administrator'
  6 = 'Production' | FR: 'Production' | EN: 'Production'
  7 = 'Configuration' | FR: 'Configuration' | EN: 'Settings'
  8 = 'Fonctions avancées' | FR: 'Fonctions avancées' | EN: 'Advanced functions'
  9 = 'Modif groupe' | FR: 'Modification du groupe' | EN: 'Group modification'
  10 = 'Creation groupe' | FR: "Création d'un groupe" | EN: 'Group creation'
   = ''
END_TEXTLIST

// ---- TextLists/TextList_Util_Userlist.TcTLO
TEXTLIST TextList_Util_Userlist
  4 = 'Liste des utilisateurs' | FR: 'Liste des utilisateurs' | EN: 'User list'
  5 = 'Liste des groupes' | FR: 'Liste des groupes' | EN: 'Group list'
  1 = 'Create user' | FR: "Création d'un nouvel utilisateur" | EN: 'New user creation'
  2 = 'user info' | FR: "Informations sur l'utilisateur" | EN: 'User information'
  3 = 'choix groupe' | FR: 'Sélection du groupe' | EN: 'Group selection'
  0 = 'Modify user' | FR: "Modification d'un utilisateur" | EN: 'User modification'
   = ''
END_TEXTLIST

// ---- TextLists/TextList_VVAT_3P.TcTLO
TEXTLIST TextList_VVAT_3P
  0 = 'ouv' | FR: 'Ouvrir' | EN: 'Open'
  1 = 'ferme' | FR: 'Fermer' | EN: 'Close'
  2 = 'lam' | FR: 'Laminer' | EN: 'Throttle'
   = ''
END_TEXTLIST

// ---- TextLists/TextList_VVAT_650_ETHERCAT.TcTLO
TEXTLIST TextList_VVAT_650_ETHERCAT
  0 = 'vanne' | FR: 'Vanne asservie' | EN: 'Servovalve'
  1 = 'max stab' | FR: 'Temps maximal de stabilisation' | EN: 'Maximum stabilization time'
  2 = 'alm stab' | FR: 'Surveillance pression - Temps avant alarme' | EN: 'Pressure supervision - Delay before alarm'
  3 = 'def stab' | FR: 'Surveillance pression - Temps avant défaut' | EN: 'Pressure supervision - Delay before fault'
  4 = 'pmin' | FR: 'Pression min. (mbar)' | EN: 'Min. pressure (mbar)'
  5 = 'pmax' | FR: 'Pression max. (mbar)' | EN: 'Max. pressure (mbar)'
  6 = 'TpsStab' | FR: 'Temps de stab.' | EN: 'Stab. time'
  7 = 'Pos' | FR: 'Position (%)' | EN: 'Position (%)'
  8 = 'Pression' | FR: 'Pression (mbar)' | EN: 'Pressure (mbar)'
   = ''
END_TEXTLIST

// ---- Visualizations/Config/Bandeaux/VISU_BANDEAU_CFG.TcVIS
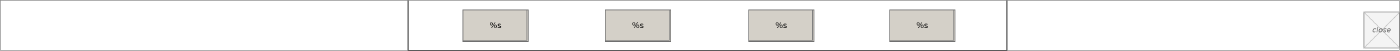
VISUALIZATION VISU_BANDEAU_CFG  // 1916x70, background image fond ecran
    Rectangle (558,0 820x70)
    Image (1866,16 50x50), image: close
        tap Global_Variables.RQ_PARAM_SYSTEM
        OnMouseClick: toggle RQ_PARAM_SYSTEM
        OnMouseClick: change screen: SYN_PROC
    Button (633,13 90x44), "%s", text list: 'TextList_Navigation', text index: 3
        OnMouseClick: change screen: VISU_CONFIG_POMPAGE
    Button (1217,13 90x44), "%s", text list: 'TextList_Navigation', text index: 4
        OnMouseClick: change screen: VISU_CONFIG_EVAP
    Button (828,13 90x44), "%s", text list: 'TextList_Navigation', text index: 8
        OnMouseClick: change screen: VISU_CONFIG_GAZ
    Button (1024,13 90x44), "%s", text list: 'TextList_Navigation', text index: 13
        OnMouseClick: change screen: VISU_CONFIG_REGEN
END_VISUALIZATION

// ---- Visualizations/Config/CRYO/VISU_CONFIG_REGEN.TcVIS
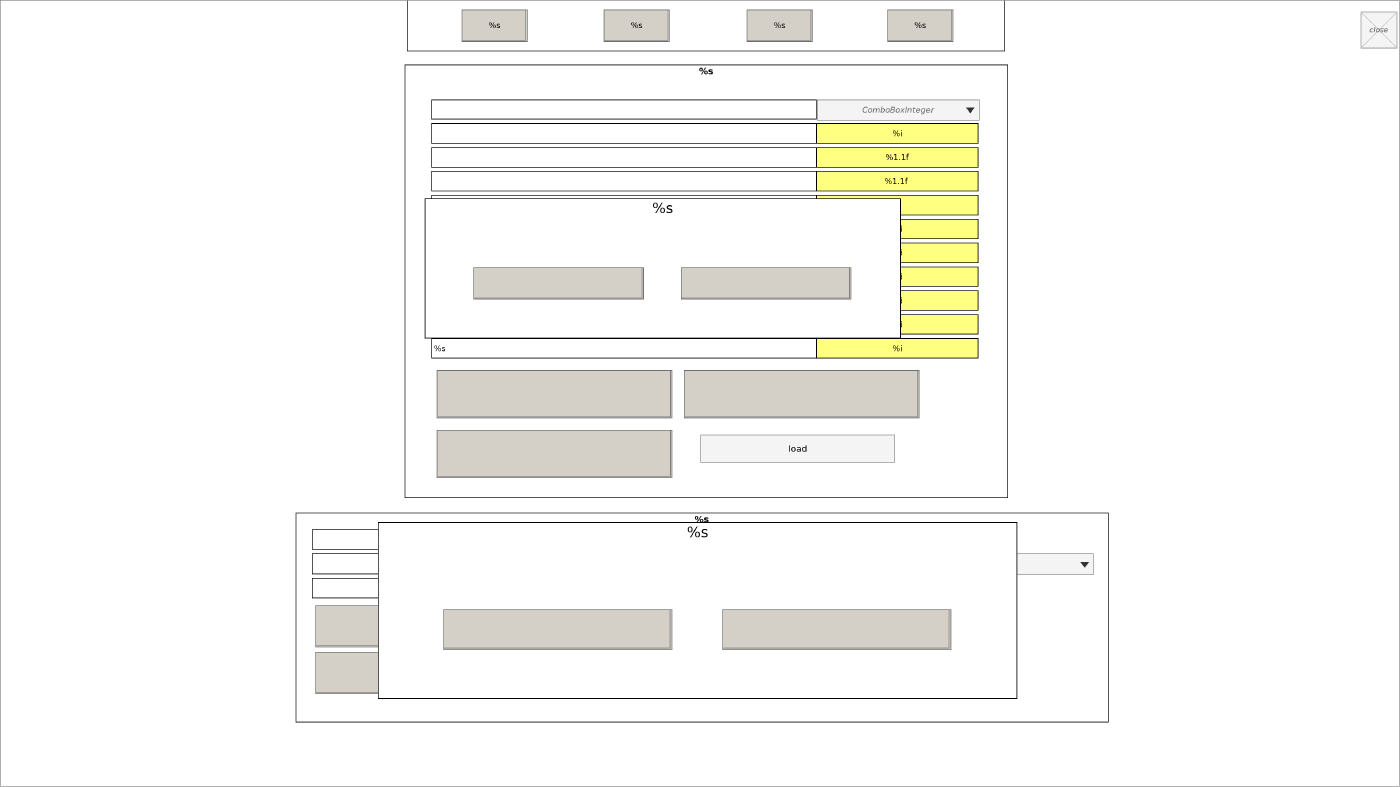
VISUALIZATION VISU_CONFIG_REGEN  // 1920x1080, background image fond_blanc_1280_1024
    Frame (0,0 1920x77)
        shows VISU_BANDEAU_CFG()
    Frame (535,82 847x601)
        shows VISU_REGENERATION(COM := PRG_POMPAGE.COM_CRYOS)
    Frame (398,687 1122x304)
        shows VISU_PARAMETRAGE_RELAY(COM := PRG_POMPAGE.COM_CRYOS)
END_VISUALIZATION

// ---- Visualizations/Config/ECOMODE/VISU_CONFIG_ECOMODE.TcVIS
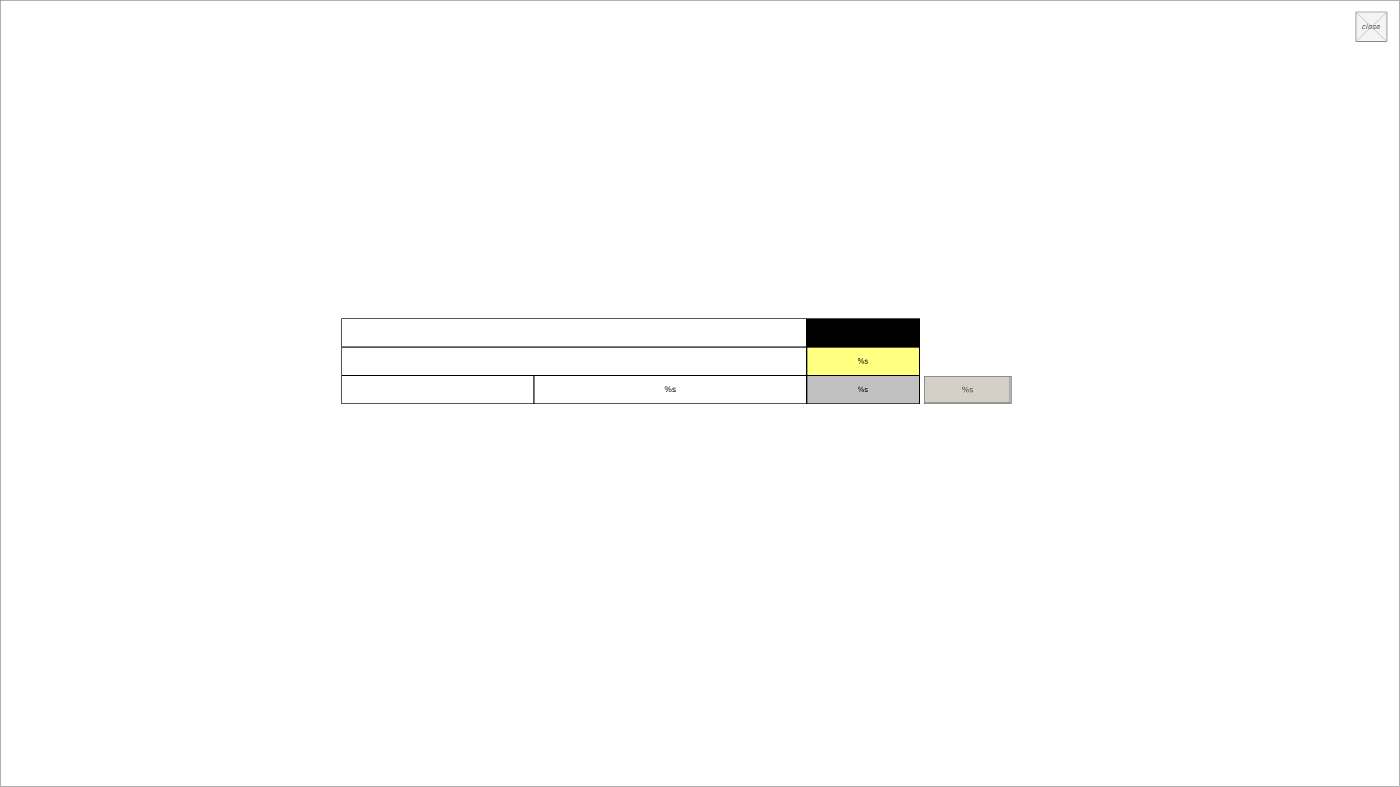
VISUALIZATION VISU_CONFIG_ECOMODE  // 1920x1080, background image fond_blanc_1280_1024
    Rectangle (468,476 638x39), text list: 'TextList_EcoMode', text index: 1
    Rectangle (468,437 638x39), text list: 'TextList_EcoMode', text index: 0
    Rectangle (468,515 264x39), text list: 'TextList_EcoMode', text index: 2
    Rectangle (1106,476 155x39), "%s", text variable: .MACHINE.CONF_Tps_Inactivite, input disabled if: NOT Global_Variables.PRG_USER.ACTU_USER.CONF_MACHINE
        OnMouseClick: write the text variable via InputWithLimits, min 0
    Rectangle (1106,437 155x39), colour toggle: MACHINE.CONF_Standby_Auto, input disabled if: NOT Global_Variables.PRG_USER.ACTU_USER.CONF_MACHINE
        toggle MACHINE.CONF_Standby_Auto
    Rectangle (732,515 374x39), "%s", text variable: .MACHINE.PRM_PROCESS_WEEKEND
    Rectangle (1106,515 155x39), "%s", colour toggle: MACHINE.PRM_RECORD_WEEKEND, text list: 'TextList_EcoMode', text index: 3
    Button (1267,516 120x38), "%s", input disabled if: NOT Global_Variables.PRG_USER.ACTU_USER.CONF_MACHINE, text list: 'TextList_EcoMode', text index: 4
        tap MAIN.bStartVerif
        OnMouseClick: execute { .MACHINE.PRM_LAUNCHER_WEEKEND:=TRUE; }
    Image (1859,16 43x41), image: close
        tap Global_Variables.RQ_PARAM_SYSTEM
        OnMouseClick: toggle RQ_PARAM_SYSTEM
        OnMouseClick: change screen: SYN_PROC
END_VISUALIZATION

// ---- Visualizations/Config/EFFLUVAGE/VISU_CONFIG_EFFLUV.TcVIS
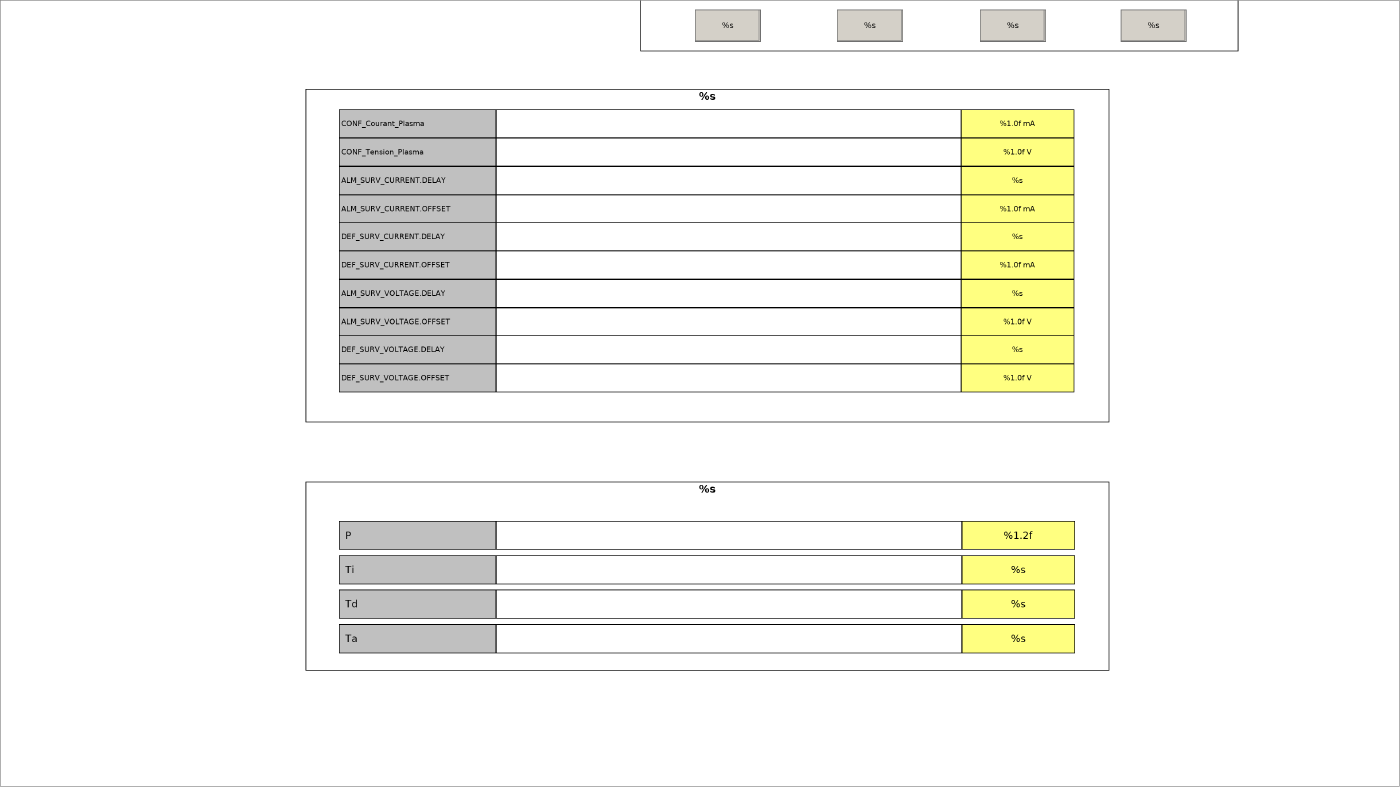
VISUALIZATION VISU_CONFIG_EFFLUV  // 1920x1080, background image fond_blanc_1280_1024
    Frame (320,0 1280x77)
        shows VISU_BANDEAU_CFG()
    RoundedRectangle (419,122 1102x457), "%s", text list: 'TextList_Config_EFFLUVAGE', text index: 0
    Rectangle (465,150 215x39), "CONF_Courant_Plasma"
    Rectangle (680,150 638x39), text list: 'TextList_Config_EFFLUVAGE', text index: 8
    Rectangle (1318,150 155x39), "%1.0f mA", text variable: PRG_EFFLUVAGE.Effluvage.ALEFF.CONF_Courant_Plasma, input disabled if: NOT Global_Variables.PRG_USER.ACTU_USER.CONF_MACHINE
        OnMouseClick: write the text variable via InputWithLimits, min 0, max 100
    Rectangle (465,189 215x39), "CONF_Tension_Plasma"
    Rectangle (680,189 638x39), text list: 'TextList_Config_EFFLUVAGE', text index: 9
    Rectangle (1318,189 155x39), "%1.0f V", text variable: PRG_EFFLUVAGE.Effluvage.ALEFF.CONF_Tension_Plasma, input disabled if: NOT Global_Variables.PRG_USER.ACTU_USER.CONF_MACHINE
        OnMouseClick: write the text variable via InputWithLimits, min 0, max 100
    Rectangle (465,228 215x39), "ALM_SURV_CURRENT.DELAY"
    Rectangle (680,228 638x39), text list: 'TextList_Config_EFFLUVAGE', text index: 11
    Rectangle (1318,228 155x39), "%s", text variable: PRG_EFFLUVAGE.Effluvage.ALEFF.ALM_Surv_Current.DELAY, input disabled if: NOT Global_Variables.PRG_USER.ACTU_USER.CONF_MACHINE
        OnMouseClick: write the text variable via InputWithLimits, min 0
    Rectangle (465,267 215x39), "ALM_SURV_CURRENT.OFFSET"
    Rectangle (680,267 638x39), text list: 'TextList_Config_EFFLUVAGE', text index: 12
    Rectangle (1318,267 155x39), "%1.0f mA", text variable: PRG_EFFLUVAGE.Effluvage.ALEFF.VAR_ALM_SURV_CURRENT.OFFSET, input disabled if: NOT Global_Variables.PRG_USER.ACTU_USER.CONF_MACHINE
        OnMouseClick: write the text variable via InputWithLimits, min 0, max 100
    Rectangle (465,305 215x39), "DEF_SURV_CURRENT.DELAY"
    Rectangle (680,305 638x39), text list: 'TextList_Config_EFFLUVAGE', text index: 13
    Rectangle (1318,305 155x39), "%s", text variable: PRG_EFFLUVAGE.Effluvage.ALEFF.DEF_Surv_Current.DELAY, input disabled if: NOT Global_Variables.PRG_USER.ACTU_USER.CONF_MACHINE
        OnMouseClick: write the text variable via InputWithLimits, min 0
    Rectangle (465,344 215x39), "DEF_SURV_CURRENT.OFFSET"
    Rectangle (680,344 638x39), text list: 'TextList_Config_EFFLUVAGE', text index: 14
    Rectangle (1318,344 155x39), "%1.0f mA", text variable: PRG_EFFLUVAGE.Effluvage.ALEFF.VAR_DEF_SURV_CURRENT.OFFSET, input disabled if: NOT Global_Variables.PRG_USER.ACTU_USER.CONF_MACHINE
        OnMouseClick: write the text variable via InputWithLimits, min 0, max 100
    RoundedRectangle (419,661 1102x259), "%s", text list: 'TextList_Config_EFFLUVAGE', text index: 0
    Frame (465,715 1009x181)
        shows VISU_CONFIG_EFF(m_Input_PRG_EFFLUVAGE := PRG_EFFLUVAGE)
    Rectangle (465,383 215x39), "ALM_SURV_VOLTAGE.DELAY"
    Rectangle (680,383 638x39), text list: 'TextList_Config_EFFLUVAGE', text index: 11
    Rectangle (1318,383 155x39), "%s", text variable: PRG_EFFLUVAGE.Effluvage.ALEFF.ALM_Surv_Voltage.DELAY, input disabled if: NOT Global_Variables.PRG_USER.ACTU_USER.CONF_MACHINE
        OnMouseClick: write the text variable via InputWithLimits, min 0
    Rectangle (465,422 215x39), "ALM_SURV_VOLTAGE.OFFSET"
    Rectangle (680,422 638x39), text list: 'TextList_Config_EFFLUVAGE', text index: 12
    Rectangle (1318,422 155x39), "%1.0f V", text variable: PRG_EFFLUVAGE.Effluvage.ALEFF.VAR_ALM_SURV_VOLTAGE.OFFSET, input disabled if: NOT Global_Variables.PRG_USER.ACTU_USER.CONF_MACHINE
        OnMouseClick: write the text variable via InputWithLimits, min 0, max 100
    Rectangle (465,460 215x39), "DEF_SURV_VOLTAGE.DELAY"
    Rectangle (680,460 638x39), text list: 'TextList_Config_EFFLUVAGE', text index: 13
    Rectangle (1318,460 155x39), "%s", text variable: PRG_EFFLUVAGE.Effluvage.ALEFF.DEF_Surv_Voltage.DELAY, input disabled if: NOT Global_Variables.PRG_USER.ACTU_USER.CONF_MACHINE
        OnMouseClick: write the text variable via InputWithLimits, min 0
    Rectangle (465,499 215x39), "DEF_SURV_VOLTAGE.OFFSET"
    Rectangle (680,499 638x39), text list: 'TextList_Config_EFFLUVAGE', text index: 14
    Rectangle (1318,499 155x39), "%1.0f V", text variable: PRG_EFFLUVAGE.Effluvage.ALEFF.VAR_DEF_SURV_VOLTAGE.OFFSET, input disabled if: NOT Global_Variables.PRG_USER.ACTU_USER.CONF_MACHINE
        OnMouseClick: write the text variable via InputWithLimits, min 0, max 100
END_VISUALIZATION

// ---- Visualizations/Config/EVAP/VISU_CONFIG_EVAP.TcVIS
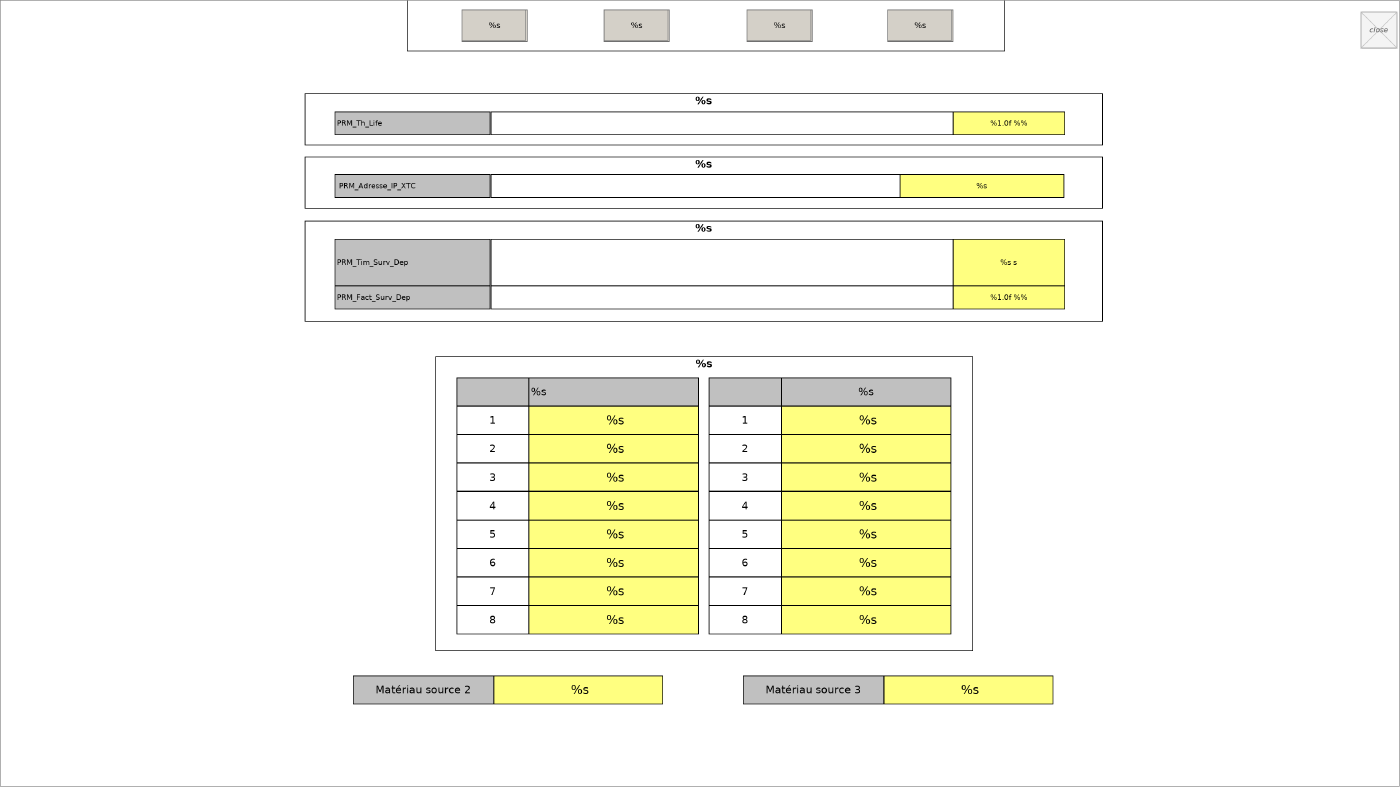
VISUALIZATION VISU_CONFIG_EVAP  // 1920x1080, background image fond_blanc_1280_1024
    Frame (0,0 1920x77)
        shows VISU_BANDEAU_CFG()
    RoundedRectangle (597,489 737x404), "%s", text list: 'TextList_Config_Evap', text index: 5
    RoundedRectangle (418,215 1094x71), "%s", text list: 'TextList_Config_Evap', text index: 20
    RoundedRectangle (418,128 1094x71), "%s", text list: 'TextList_Config_Evap', text index: 0
    Group (459,153 1001x32)
        Rectangle (214,0 634x32), text list: 'TextList_Config_Evap', text index: 1
        Rectangle (848,0 153x32), "%1.0f %%", text variable: PRG_EVAP.PRM_Seuil_Crystal_Life, input disabled if: NOT Global_Variables.PRG_USER.ACTU_USER.CONF_MACHINE
            OnMouseClick: write the text variable via InputWithLimits, min 0, max 100
        Rectangle (0,0 213x32), "PRM_Th_Life"
    RoundedRectangle (418,303 1094x138), "%s", text list: 'TextList_Config_Evap', text index: 2
    Rectangle (673,328 634x64), text list: 'TextList_Config_Evap', text index: 3
    Rectangle (1307,328 153x64), "%s s", text variable: PRG_EVAP.EVAPS1.PRM_TPS_MIN_SURV_DEPOT, input disabled if: NOT Global_Variables.PRG_USER.ACTU_USER.CONF_MACHINE
        OnMouseClick: write the text variable via InputWithLimits, min 0
    Rectangle (459,328 213x64), "PRM_Tim_Surv_Dep"
    Rectangle (673,392 634x32), text list: 'TextList_Config_Evap', text index: 4
    Rectangle (1307,392 153x32), "%1.0f %%", text variable: PRG_EVAP.EVAPS1.PRM_FACTEUR_TEMPS_DEPOT, input disabled if: NOT Global_Variables.PRG_USER.ACTU_USER.CONF_MACHINE
        OnMouseClick: write the text variable via InputWithLimits, min 0
    Rectangle (459,392 213x32), "PRM_Fact_Surv_Dep"
    Group (459,239 1000x32)
        Rectangle (0,0 213x32), "PRM_Adresse_IP_XTC", text variable: 1
        Rectangle (214,0 562x32), text list: 'TextList_Config_Evap', text index: 21
        Rectangle (775,0 225x32), "%s", text variable: Global_Variables.PRG_EVAP.PRM_Adresse_IP_XTC, input disabled if: NOT Global_Variables.PRG_USER.ACTU_USER.CONF_MACHINE
            OnMouseDown: write the text variable via InputWithLimits
    Frame (626,518 332x352)
        shows VISU_CONF_MAT(m_Input_CRUCIBLE := PRG_EVAP.CRUCIBLE1)
    Frame (972,518 332x352)
        shows VISU_CONF_BAL(m_Input_SWEEP := PRG_EVAP.SWEEP1)
    Rectangle (484,927 193x39), "Matériau source 2"
    Rectangle (677,927 232x39), "%s", text variable: Global_Variables.PRG_EVAP.PRM_Mat_Source2, input disabled if: NOT Global_Variables.PRG_USER.ACTU_USER.CONF_MACHINE
        OnMouseDown: write the text variable via InputWithLimits
    Rectangle (1019,927 193x39), "Matériau source 3"
    Rectangle (1212,927 232x39), "%s", text variable: Global_Variables.PRG_EVAP.PRM_Mat_Source3, input disabled if: NOT Global_Variables.PRG_USER.ACTU_USER.CONF_MACHINE
        OnMouseDown: write the text variable via InputWithLimits
END_VISUALIZATION

// ---- Visualizations/Config/GAZ/VISU_CONFIG_GAZ.TcVIS
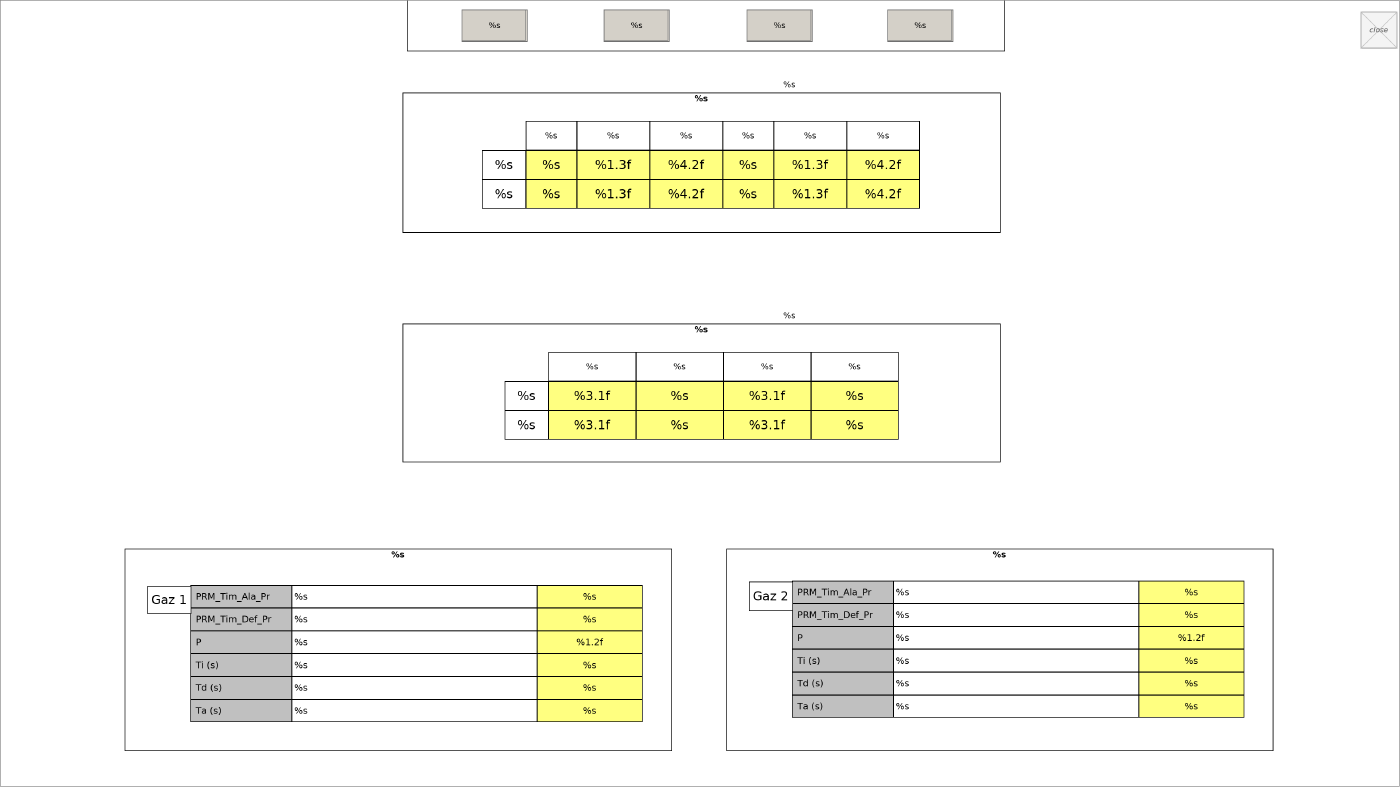
VISUALIZATION VISU_CONFIG_GAZ  // 1920x1080
    RoundedRectangle (996,753 750x277), "%s", text list: 'TextList_Config_Gaz', text index: 35
    RoundedRectangle (171,753 750x277), "%s", text list: 'TextList_Config_Gaz', text index: 35
    Frame (0,0 1920x77)
        shows VISU_BANDEAU_CFG()
    Frame (722,206 542x44)
        shows VISU_CONFIG_LIGNE_GAZ_SEUIL_MFC_MKS(m_Input_MASSFLOW := PRG_GAZ.DG[1])
    RoundedRectangle (552,127 820x192), "%s", text list: 'TextList_Config_Gaz', text index: 1
    Rectangle (1071,106 300x20), "%s", text list: 'TextList_Config_Gaz', text index: 3
    Rectangle (1071,423 300x20), "%s", text list: 'TextList_Config_Gaz', text index: 4
    RoundedRectangle (552,444 820x190), "%s", text list: 'TextList_Config_Gaz', text index: 2
    Rectangle (791,166 100x40), "%s", text list: 'TextList_Config_Gaz', text index: 6
    Rectangle (891,166 100x40), "%s", text list: 'TextList_Config_Gaz', text index: 7
    Rectangle (1161,166 100x40), "%s", text list: 'TextList_Config_Gaz', text index: 9
    Rectangle (991,166 70x40), "%s", text list: 'TextList_Config_Gaz', text index: 8
    Rectangle (1061,166 100x40), "%s", text list: 'TextList_Config_Gaz', text index: 6
    Rectangle (721,166 70x40), "%s", text list: 'TextList_Config_Gaz', text index: 5
    Rectangle (661,206 60x40), "%s", text list: 'TextList_Config_Gaz', text index: 11
    Frame (721,246 542x44)
        shows VISU_CONFIG_LIGNE_GAZ_SEUIL_MFC_MKS(m_Input_MASSFLOW := PRG_GAZ.DG[2])
    Rectangle (661,246 60x40), "%s", text list: 'TextList_Config_Gaz', text index: 12
    Frame (721,206 542x44)
        shows VISU_CONFIG_LIGNE_GAZ_SEUIL_MFC_MKS(m_Input_MASSFLOW := PRG_GAZ.DG[1])
        p1532468285: PRG_GAZ.DG[1]
    Rectangle (692,523 60x40), "%s", text list: 'TextList_Config_Gaz', text index: 11
    Rectangle (1112,483 120x40), "%s", text list: 'TextList_Config_Gaz', text index: 23
    Rectangle (872,483 120x40), "%s", text list: 'TextList_Config_Gaz', text index: 21
    Rectangle (992,483 120x40), "%s", text list: 'TextList_Config_Gaz', text index: 22
    Rectangle (752,483 120x40), "%s", text list: 'TextList_Config_Gaz', text index: 20
    Frame (752,523 479x42)
        shows VISU_CONFIG_LIGNE_GAZ_SURV_MFC_MKS(m_Input_MASSFLOW := PRG_GAZ.DG[1])
    Frame (752,563 479x42)
        shows VISU_CONFIG_LIGNE_GAZ_SURV_MFC_MKS(m_Input_MASSFLOW := PRG_GAZ.DG[2])
    Rectangle (692,563 60x40), "%s", text list: 'TextList_Config_Gaz', text index: 12
    Frame (261,803 620x200)
        shows VISU_CONFIG_REGUL_GAZ(m_Input_REGULATION := Global_Variables.PRG_GAZ.REGULATION_GAZ_L1)
    Rectangle (202,804 60x38), "Gaz 1"
    Frame (1086,797 620x200)
        shows VISU_CONFIG_REGUL_GAZ(m_Input_REGULATION := Global_Variables.PRG_GAZ.REGULATION_GAZ_L2)
    Rectangle (1027,798 60x40), "Gaz 2"
END_VISUALIZATION

// ---- Visualizations/Config/MOUVEMENTS/VISU_CONFIG_MOUVEMENTS.TcVIS
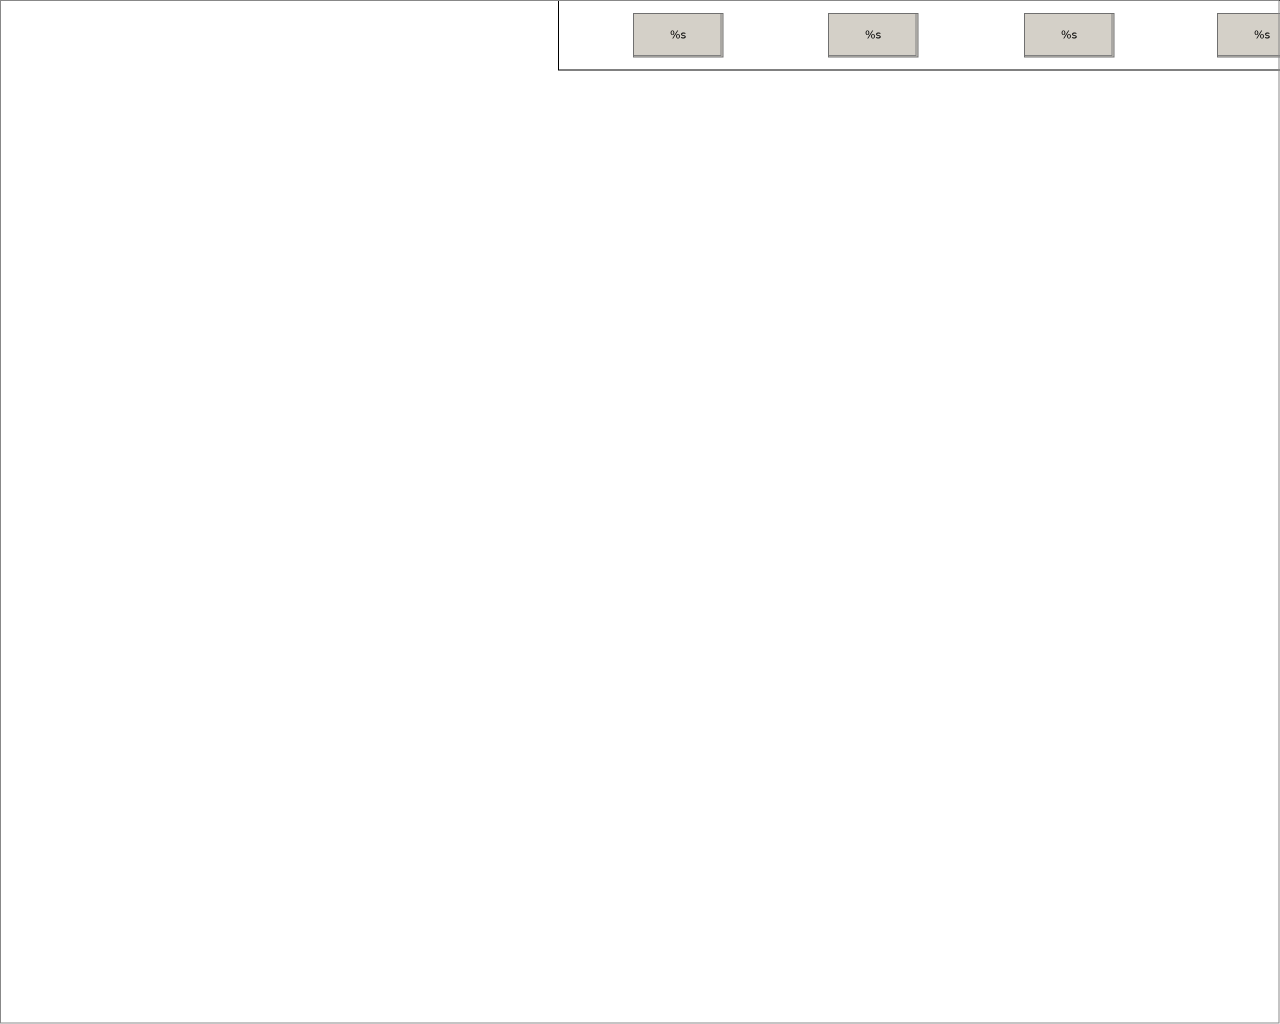
VISUALIZATION VISU_CONFIG_MOUVEMENTS  // 1280x1024, background image fond_blanc_1280_1024
    Frame (0,0 1280x77)
        shows VISU_BANDEAU_CFG()
END_VISUALIZATION

// ---- Visualizations/Config/POMPAGE/VISU_CONFIG_POMPAGE.TcVIS
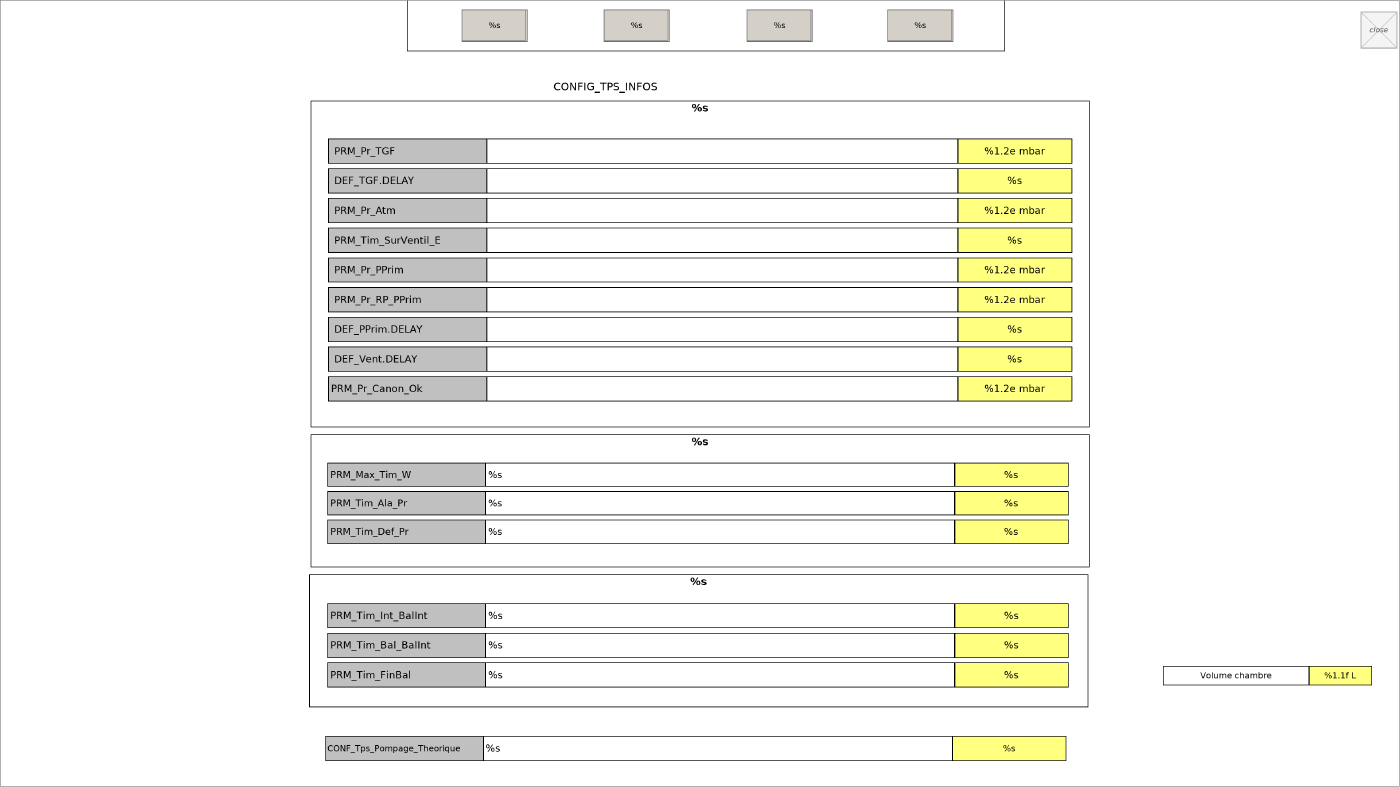
VISUALIZATION VISU_CONFIG_POMPAGE  // 1920x1080, background image fond_blanc_1280_1024
    RoundedRectangle (426,138 1068x448), "%s", text list: 'TextList_Config_Pompage', text index: 0
    Frame (0,0 1920x77)
        shows VISU_BANDEAU_CFG()
    Rectangle (756,109 300x20), "CONFIG_TPS_INFOS"
    Rectangle (1595,914 200x26), "Volume chambre"
    Rectangle (1795,914 86x26), "%1.1f L", text variable: Global_Variables.PRG_POMPAGE.POMPAGE.CONF_Volume_Enceinte, input disabled if: NOT Global_Variables.PRG_USER.ACTU_USER.CONF_MACHINE
        OnMouseDown: write the text variable via InputWithLimits
    Frame (449,189 1021x379)
        shows VISU_CONFIG_POMPAGE_CHAMBRE(m_Input_PRG_POMPAGE := PRG_POMPAGE)
    RoundedRectangle (426,596 1068x182), "%s", text list: 'TextList_Config_Pompage', text index: 15
    Rectangle (446,1010 217x34), "CONF_Tps_Pompage_Theorique"
    Rectangle (663,1010 643x34), "%s", text list: 'TextList_Config_Pompage', text index: 16
    Rectangle (1306,1010 156x34), "%s", text variable: PRG_POMPAGE.CONF_Tps_Pompage_Theorique, input disabled if: NOT Global_Variables.PRG_USER.ACTU_USER.CONF_MACHINE
        OnMouseDown: write the text variable via InputWithLimits
    RoundedRectangle (424,788 1068x182), "%s", text list: 'TextList_Config_Pompage', text index: 20
    Frame (449,828 1016x141)
        shows VISU_CONFIG_INTERJOINT(m_Input_Pompage := PRG_POMPAGE.POMPAGE)
    Frame (449,635 1016x111)
        shows VISU_CONFIG_VANNE_ASS_VVAT650(m_Input_Vanne := PRG_POMPAGE.POMPAGE.VS11)
END_VISUALIZATION

// ---- Visualizations/Semi Auto/Elements/SA_CACHE_ACTUATOR.TcVIS
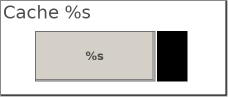
VISUALIZATION SA_CACHE_ACTUATOR  // 228x97
VAR_IN_OUT
	m_Input_PRM_Forcage : Bool;
END_VAR
VAR_INPUT
	m_Input_CACHE : BLOCK_ACTUATOR;
END_VAR
    RoundedRectangle (0,0 226x95), "Cache %s", text variable: m_Input_CACHE.MNEMO
    RoundedRectangle (157,31 30x50), colour toggle: m_Input_CACHE.STATE_ON
    Button (35,31 120x50), "%s", input disabled if: NOT (PRG_User.ACTU_USER.FONCTION_SA AND NOT MACHINE.STATE_PROD), text list: 'TextList_Orders', text index: 0
        toggle m_Input_PRM_Forcage
END_VISUALIZATION

// ---- Visualizations/Semi Auto/Elements/SA_CACHE_ACTUATOR2.TcVIS
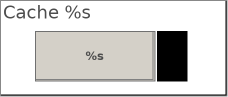
VISUALIZATION SA_CACHE_ACTUATOR2  // 228x97
VAR_IN_OUT
	m_Input_PRM_Forcage : Bool;
END_VAR
VAR_INPUT
	m_Input_CACHE : BLOCK_ACTUATOR2;
END_VAR
    RoundedRectangle (0,0 226x95), "Cache %s", text variable: m_Input_CACHE.MNEMO
    RoundedRectangle (157,31 30x50), colour toggle: m_Input_CACHE.STATE_ON
    Button (35,31 120x50), "%s", input disabled if: NOT (PRG_User.ACTU_USER.FONCTION_SA AND NOT MACHINE.STATE_PROD), text list: 'TextList_Orders', text index: 0
        toggle m_Input_PRM_Forcage
END_VISUALIZATION

// ---- Visualizations/Semi Auto/Elements/SA_EFFLUVAGE.TcVIS
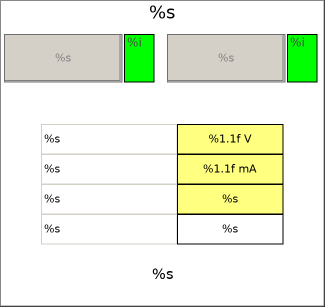
VISUALIZATION SA_EFFLUVAGE  // 325x307
VAR_IN_OUT
	m_input_effluvage:		BLOCK_PRG_EFFLUVAGE;
	m_Input_Machine:		BLOCK_MODE_MARCHE_V2_0;
END_VAR
    RoundedRectangle (0,0 325x307), "%s", text list: 'TextList_Effluvage', text index: 1
    Frame (4,34 152x50)
        shows VISU_FCTS_SA(m_Input_ID_XML := 29, m_Input_Operation := m_input_effluvage.Effluvage.OP_Marche_Eff, m_Input_UserRight := PRG_USER.ACTU_USER.FONCTION_SA)
    Frame (167,34 152x50)
        shows VISU_FCTS_SA(m_Input_ID_XML := 7, m_Input_Operation := m_input_effluvage.Effluvage.OP_Arret_Eff, m_Input_UserRight := PRG_USER.ACTU_USER.FONCTION_SA)
    Textfield (41,154 136x30), "%s", text list: 'TextList_Effluvage', text index: 2
    Textfield (41,184 136x30), "%s", text list: 'TextList_Effluvage', text index: 3
    Rectangle (177,154 106x30), "%1.1f mA", text variable: m_input_effluvage.Effluvage.PRM_consigne, input disabled if: (NOT PRG_User.ACTU_USER.MAINTENANCE AND NOT PRG_User.ACTU_USER.FONCTION_SA AND NOT PRG_User.ACTU_USER.MODIF_ENLIGNE) OR (NOT MACHINE.STATE_Wait_Prod AND NOT MACHINE.STATE_Manu)
        OnMouseClick: write the text variable via InputWithLimits, min 0
    Rectangle (177,184 106x30), "%s", text variable: m_input_effluvage.Effluvage.PRM_TPS_effluvage, input disabled if: (NOT PRG_User.ACTU_USER.MAINTENANCE AND NOT PRG_User.ACTU_USER.FONCTION_SA AND NOT PRG_User.ACTU_USER.MODIF_ENLIGNE) OR (NOT MACHINE.STATE_Wait_Prod AND NOT MACHINE.STATE_Manu)
        OnMouseClick: write the text variable via InputWithLimits, min 0
    Textfield (41,214 136x30), "%s", text list: 'TextList_Effluvage', text index: 4
    Rectangle (177,214 106x30), "%s", text variable: m_input_effluvage.Effluvage.TIMER_Effluvage.ET, input disabled if: (NOT PRG_User.ACTU_USER.MAINTENANCE AND NOT PRG_User.ACTU_USER.FONCTION_SA AND NOT PRG_User.ACTU_USER.MODIF_ENLIGNE) OR (NOT MACHINE.STATE_Wait_Prod AND NOT MACHINE.STATE_Manu)
    Rectangle (42,259 242x30), "%s", text variable: PRG_EFFLUVAGE.Effluvage.TIMER_Effluvage.ET, invisible if: Not PRG_EFFLUVAGE.Effluvage.OP_Marche_Eff.Etape.3, text list: 'TextList_Gaz', text index: 4
    Textfield (41,124 136x30), "%s", text list: 'TextList_Effluvage', text index: 5
    Rectangle (177,124 106x30), "%1.1f V", text variable: m_input_effluvage.Effluvage.PRM_Tension_attendue, input disabled if: (NOT PRG_User.ACTU_USER.MAINTENANCE AND NOT PRG_User.ACTU_USER.FONCTION_SA AND NOT PRG_User.ACTU_USER.MODIF_ENLIGNE) OR (NOT MACHINE.STATE_Wait_Prod AND NOT MACHINE.STATE_Manu)
        OnMouseClick: write the text variable via InputWithLimits, min 0
END_VISUALIZATION

// ---- Visualizations/Semi Auto/Elements/SA_EVAP.TcVIS
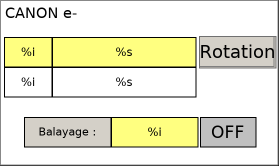
VISUALIZATION SA_EVAP  // 279x166
VAR_IN_OUT
	m_Input_Crucible:   BLOCK_IND_CR_396_TELEMARK;
	m_Input_Sweep:		BLOCK_TELEMARK_CHEETAH_SWEEP;	
END_VAR
    RoundedRectangle (0,0 279x166), text variable: m_Input_Crucible.MNEMO
    Rectangle (2,1 104x24), "CANON e-"
    Rectangle (111,117 87x30), "%i", text variable: m_Input_Sweep.PRM_NbBal, input disabled if: NOT (Global_Variables.PRG_USER.ACTU_USER.FONCTION_SA AND NOT MACHINE.STATE_PROD)
        OnMouseClick: write the text variable via InputWithLimits, min 1, max 8
    Rectangle (24,117 87x30), "Balayage :"
    Rectangle (4,37 48x30), "%i", text variable: m_Input_Crucible.PRM_NCR, input disabled if: NOT (Global_Variables.PRG_USER.ACTU_USER.FONCTION_SA AND NOT MACHINE.STATE_PROD)
        OnMouseClick: write the text variable via InputWithLimits, min 1, max m_Input_Crucible.CONF_NCR
    Rectangle (52,37 144x30), "%s", text variable: m_Input_Crucible.PRM_MAT[m_Input_Crucible.PRM_NCR]
    Button (199,36 77x32), "Rotation", input disabled if: NOT (PRG_USER.ACTU_USER.FONCTION_SA AND NOT MACHINE.STATE_Prod)
        tap PRG_EVAP.PRM_Forcage_Crucible
    RoundedRectangle (200,117 56x30), "ON", invisible if: NOT m_Input_Sweep.STATE_ON
    RoundedRectangle (200,117 56x30), "OFF", invisible if: NOT m_Input_Sweep.STATE_OFF
    Rectangle (4,67 48x30), "%i", text variable: m_Input_Crucible.STATE_POS
    Rectangle (52,67 144x30), "%s", text variable: m_Input_Crucible.PRM_MAT[m_Input_Crucible.STATE_POS], invisible if: (m_Input_Crucible.STATE_POS < 1) or (m_Input_Crucible.STATE_POS > m_Input_Crucible.CONF_NCR)
END_VISUALIZATION

// ---- Visualizations/Semi Auto/Elements/SA_HEATING.TcVIS
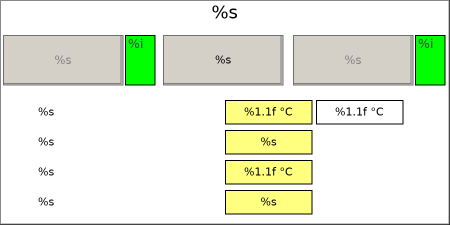
VISUALIZATION SA_HEATING  // 450x225
VAR_IN_OUT
	m_Input_UserRight:	BOOL;
	m_Input_Machine:	BLOCK_MODE_MARCHE_V2_0;
	m_Input_PRG:		BLOCK_PRG_CHAUFFAGE;
END_VAR
    Rectangle (0,0 450x225), "%s", text list: 'TextList_Navigation', text index: 10
    Frame (3,35 153x52)
        shows VISU_FCTS_SA(m_Input_ID_XML := 24, m_Input_UserRight := PRG_USER.ACTU_USER.FONCTION_SA, m_Input_Operation := m_Input_PRG.CHAUFFAGE.OP_MARCHE)
    Frame (293,35 153x52)
        shows VISU_FCTS_SA(m_Input_ID_XML := 25, m_Input_UserRight := PRG_USER.ACTU_USER.FONCTION_SA, m_Input_Operation := m_Input_PRG.CHAUFFAGE.OP_ARRET)
    Button (163,35 120x50), "%s", input disabled if: (NOT PRG_USER.ACTU_USER.FONCTION_SA AND NOT m_Input_Machine.STATE_Prod) OR (NOT PRG_USER.ACTU_USER.MODIF_ENLIGNE AND m_Input_Machine.STATE_Prod), text list: 'TextList_Basiques', text index: 19
        tap m_Input_PRG.CHAUFFAGE.CO_Modif
    Rectangle (35,100 188x24), "%s", text list: 'TextList_Chauffage', text index: 9
    RoundedRectangle (316,100 87x24), "%1.1f °C", text variable: m_Input_PRG.CHAUFFAGE.CH.IN_Temperature
    RoundedRectangle (225,100 87x24), "%1.1f °C", text variable: m_Input_PRG.CHAUFFAGE.PRM_Temp, input disabled if: (NOT PRG_USER.ACTU_USER.FONCTION_SA AND NOT m_Input_Machine.STATE_Prod) OR (NOT PRG_USER.ACTU_USER.MODIF_ENLIGNE AND m_Input_Machine.STATE_Prod)
        OnMouseClick: write the text variable via VisuDialogs.Numpad, min 20, max m_Input_PRG.PRM_Max_Temp
    Rectangle (35,130 188x24), "%s", text list: 'TextList_Chauffage', text index: 6
    RoundedRectangle (225,130 87x24), "%s", text variable: m_Input_PRG.CHAUFFAGE.PRM_Tps_Stab, input disabled if: (NOT PRG_USER.ACTU_USER.FONCTION_SA AND NOT m_Input_Machine.STATE_Prod) OR (NOT PRG_USER.ACTU_USER.MODIF_ENLIGNE AND m_Input_Machine.STATE_Prod)
        OnMouseClick: write the text variable via VisuDialogs.Keypad
    Rectangle (35,160 188x24), "%s", text list: 'TextList_Chauffage', text index: 10
    RoundedRectangle (225,160 87x24), "%1.1f °C", text variable: m_Input_PRG.CHAUFFAGE.PRM_Delta_Stab, input disabled if: (NOT PRG_USER.ACTU_USER.FONCTION_SA AND NOT m_Input_Machine.STATE_Prod) OR (NOT PRG_USER.ACTU_USER.MODIF_ENLIGNE AND m_Input_Machine.STATE_Prod)
        OnMouseClick: write the text variable via VisuDialogs.Numpad, min 0, max 50
    Rectangle (35,190 188x24), "%s", text list: 'TextList_Chauffage', text index: 8
    RoundedRectangle (225,190 87x24), "%s", text variable: m_Input_PRG.CHAUFFAGE.DEF_Stab.DELAY, input disabled if: (NOT PRG_USER.ACTU_USER.FONCTION_SA AND NOT m_Input_Machine.STATE_Prod) OR (NOT PRG_USER.ACTU_USER.MODIF_ENLIGNE AND m_Input_Machine.STATE_Prod)
        OnMouseClick: write the text variable via VisuDialogs.Keypad
END_VISUALIZATION

// ---- Visualizations/Semi Auto/Elements/SA_IAD.TcVIS
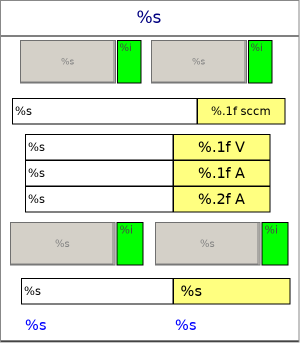
VISUALIZATION SA_IAD  // 300x343
VAR_IN_OUT
	m_Input_CANON_ION : BLOCK_CANON_ION_MARK3;
	m_Input_IAD : BLOCK_MARK3_PLUS;
END_VAR
    Rectangle (-1,-2 300x343)
    Rectangle (25,134 148x26), "%s", text list: 'TextList_IAD', text index: 0
    Rectangle (173,134 97x26), "%.1f V", text variable: m_Input_IAD.PRM_ANODE_VOLTAGE, input disabled if: ((NOT PRG_User.ACTU_USER.MAINTENANCE AND NOT PRG_User.ACTU_USER.FONCTION_SA AND NOT PRG_User.ACTU_USER.MODIF_ENLIGNE) OR (NOT MACHINE.STATE_Wait_Prod AND NOT MACHINE.STATE_Manu)) <> 0
        OnMouseDown: write the text variable via VisuDialogs.Numpad, min 0, max 300
    Rectangle (21,278 152x26), "%s", text list: 'TextList_IAD', text index: 11
    Rectangle (173,278 117x26), "%s", text variable: m_Input_CANON_ION.PRM_TPS_IAD, input disabled if: ((NOT PRG_User.ACTU_USER.MAINTENANCE AND NOT PRG_User.ACTU_USER.FONCTION_SA AND NOT PRG_User.ACTU_USER.MODIF_ENLIGNE) OR (NOT MACHINE.STATE_Wait_Prod AND NOT MACHINE.STATE_Manu)) <> 0
        OnMouseDown: write the text variable via VisuDialogs.Keypad
    Rectangle (172,312 117x26), "%s", text variable: m_Input_CANON_ION.STATE_IAD, invisible if: NOT m_Input_CANON_ION.OP_IAD.Etape.3
    Rectangle (25,186 148x26), "%s", text list: 'TextList_IAD', text index: 2
    Rectangle (173,186 97x26), "%.2f A", text variable: m_Input_IAD.PRM_NEUTRAL_CURRENT, input disabled if: ((NOT PRG_User.ACTU_USER.MAINTENANCE AND NOT PRG_User.ACTU_USER.FONCTION_SA AND NOT PRG_User.ACTU_USER.MODIF_ENLIGNE) OR (NOT MACHINE.STATE_Wait_Prod AND NOT MACHINE.STATE_Manu)) <> 0
        OnMouseDown: write the text variable via VisuDialogs.Numpad, min 0, max 1.86
    Rectangle (25,160 148x26), "%s", text list: 'TextList_IAD', text index: 1
    Rectangle (173,160 97x26), "%.1f A", text variable: m_Input_IAD.PRM_ANODE_CURRENT, input disabled if: ((NOT PRG_User.ACTU_USER.MAINTENANCE AND NOT PRG_User.ACTU_USER.FONCTION_SA AND NOT PRG_User.ACTU_USER.MODIF_ENLIGNE) OR (NOT MACHINE.STATE_Wait_Prod AND NOT MACHINE.STATE_Manu)) <> 0
        OnMouseDown: write the text variable via VisuDialogs.Numpad, min 0, max 15
    Rectangle (-1,-2 300x38), "%s", text list: 'TextList_IAD', text index: 10
    Rectangle (22,312 147x26), "%s", invisible if: NOT m_Input_CANON_ION.OP_IAD.Etape.3, text list: 'TextList_IAD'
    Rectangle (12,98 185x26), "%s", text list: 'TextList_IAD', text index: 8
    Rectangle (197,98 88x26), "%.1f sccm", text variable: m_Input_CANON_ION.PRM_GAZ_1C_AMORCAGE, input disabled if: ((NOT PRG_User.ACTU_USER.MAINTENANCE AND NOT PRG_User.ACTU_USER.FONCTION_SA AND NOT PRG_User.ACTU_USER.MODIF_ENLIGNE) OR (NOT MACHINE.STATE_Wait_Prod AND NOT MACHINE.STATE_Manu)) <> 0
        OnMouseDown: write the text variable via VisuDialogs.Numpad, min 0, max 100
    Frame (151,40 123x45)
        shows VISU_FCTS_SA(m_Input_ID_XML := 7, m_Input_UserRight := PRG_USER.ACTU_USER.FONCTION_SA, m_Input_Operation := m_Input_CANON_ION.OP_ARRET)
    Frame (20,40 123x45)
        shows VISU_FCTS_SA(m_Input_ID_XML := 5, m_Input_UserRight := PRG_USER.ACTU_USER.FONCTION_SA, m_Input_Operation := m_Input_CANON_ION.OP_MARCHE)
    Frame (155,222 135x45)
        shows VISU_FCTS_SA(m_Input_ID_XML := 27, m_Input_UserRight := PRG_USER.ACTU_USER.FONCTION_SA, m_Input_Operation := m_Input_CANON_ION.OP_STOP_IAD)
    Frame (10,222 135x45)
        shows VISU_FCTS_SA(m_Input_ID_XML := 26, m_Input_UserRight := PRG_USER.ACTU_USER.FONCTION_SA, m_Input_Operation := m_Input_CANON_ION.OP_IAD)
END_VISUALIZATION

// ---- Visualizations/Semi Auto/Elements/SA_LIGNE_GAZ_ANA_RAMPE.TcVIS
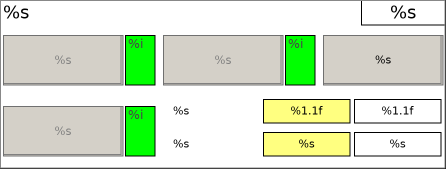
VISUALIZATION SA_LIGNE_GAZ_ANA_RAMPE  // 446x169
VAR_IN_OUT
	m_Input_Ligne:		BLOCK_LIGNE_GAZ;
	m_Input_Machine:	BLOCK_MODE_MARCHE_V2_0;
	m_Input_DG:			BLOCK_MFC_ANA2;
	m_Input_UserRight:	BOOL;
END_VAR

VAR_INPUT
	m_Input_NumTextList:		INT;
END_VAR
    Rectangle (0,0 446x169), "%s", text list: 'TextList_Gaz', text index: m_Input_NumTextList
    Rectangle (361,0 85x25), "%s", text variable: m_Input_DG.CONF_Util_Name
    Frame (3,35 153x52)
        shows VISU_FCTS_SA(m_Input_ID_XML := 12, m_Input_UserRight := PRG_USER.ACTU_USER.FONCTION_SA AND NOT m_Input_Machine.STATE_Prod, m_Input_Operation := m_Input_Ligne.OP_MARCHE)
    Frame (3,106 153x52)
        shows VISU_FCTS_SA(m_Input_ID_XML := 13, m_Input_UserRight := PRG_USER.ACTU_USER.FONCTION_SA AND NOT m_Input_Machine.STATE_Prod, m_Input_Operation := m_Input_Ligne.OP_ARRET)
    Rectangle (170,99 91x24), "%s", text list: 'TextList_Gaz', text index: 3
    RoundedRectangle (354,99 87x24), "%1.1f", text variable: m_Input_DG.STATE_Flow
    RoundedRectangle (263,99 87x24), "%1.1f", text variable: m_Input_Ligne.PRM_Flow, input disabled if: (NOT PRG_USER.ACTU_USER.FONCTION_SA AND NOT m_Input_Machine.STATE_Prod) OR (NOT PRG_USER.ACTU_USER.MODIF_ENLIGNE AND m_Input_Machine.STATE_Prod)
        OnMouseClick: write the text variable via VisuDialogs.Numpad, min 0, max m_Input_DG.CONF_Util_Max_Flow
    Rectangle (170,132 91x24), "%s", text list: 'TextList_Basiques', text index: 22
    RoundedRectangle (263,132 87x24), "%s", text variable: m_Input_Ligne.OP_RAMPE.PRM_Temps, input disabled if: (NOT PRG_USER.ACTU_USER.FONCTION_SA AND NOT m_Input_Machine.STATE_Prod) OR (NOT PRG_USER.ACTU_USER.MODIF_ENLIGNE AND m_Input_Machine.STATE_Prod)
        OnMouseClick: write the text variable via VisuDialogs.Keypad
    Frame (163,35 153x52)
        shows VISU_FCTS_SA(m_Input_ID_XML := 14, m_Input_UserRight := PRG_USER.ACTU_USER.FONCTION_SA AND NOT m_Input_Machine.STATE_Prod, m_Input_Operation := m_Input_Ligne.OP_RAMPE.MARCHE)
    Button (323,35 120x50), "%s", input disabled if: (NOT PRG_USER.ACTU_USER.FONCTION_SA AND NOT m_Input_Machine.STATE_Prod) OR (NOT PRG_USER.ACTU_USER.MODIF_ENLIGNE AND m_Input_Machine.STATE_Prod), text list: 'TextList_Basiques', text index: 19
        toggle m_Input_Ligne.CO_Modif
    RoundedRectangle (354,132 87x24), "%s", text variable: m_Input_Ligne.OP_RAMPE.OUT_Tps_ecoule
END_VISUALIZATION

// ---- Visualizations/Semi Auto/Elements/SA_LIGNE_GAZ_BROOKS_RAMPE.TcVIS
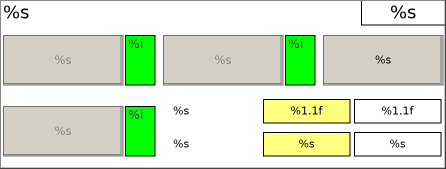
VISUALIZATION SA_LIGNE_GAZ_BROOKS_RAMPE  // 446x169
VAR_IN_OUT
	m_Input_Ligne:		BLOCK_LIGNE_GAZ;
	m_Input_Machine:	BLOCK_MODE_MARCHE_V2_0;
	m_Input_DG:			BLOCK_MFC_BROOKS_NoCoE;
	m_Input_UserRight:	BOOL;
END_VAR

